REGION Network 4: Set drive objects for drive diagnostic
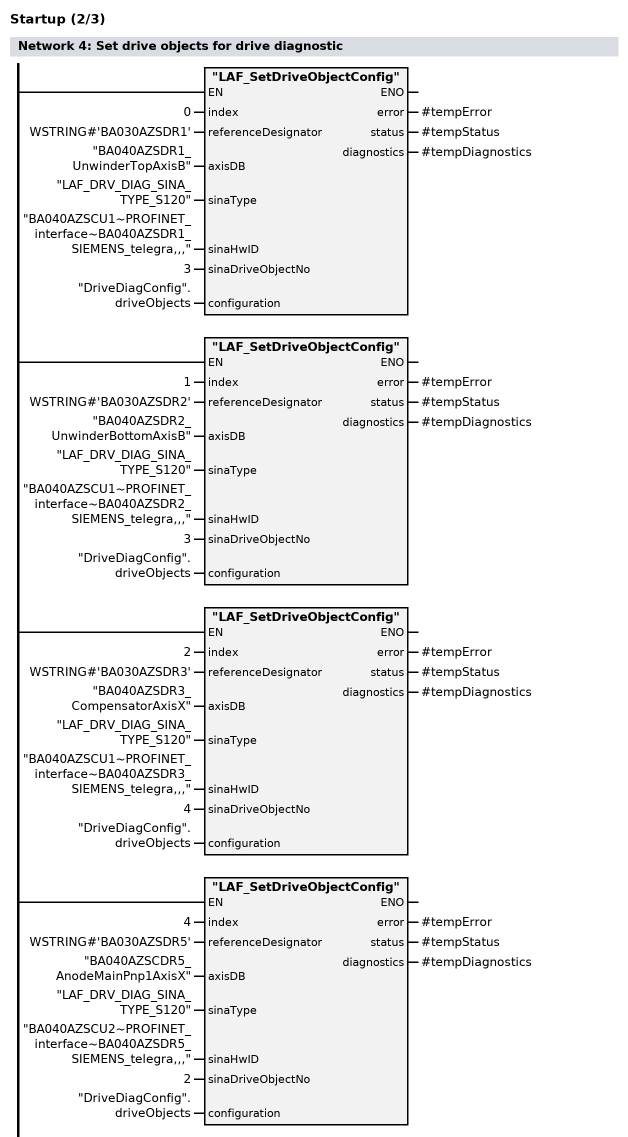
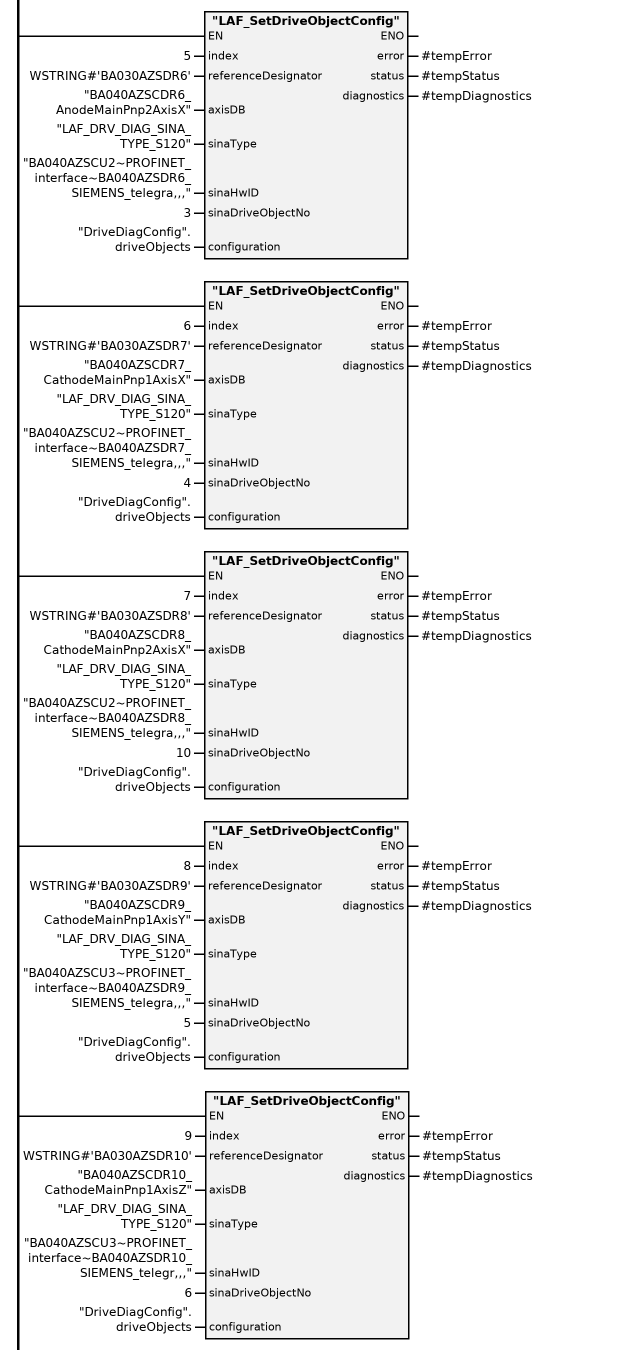
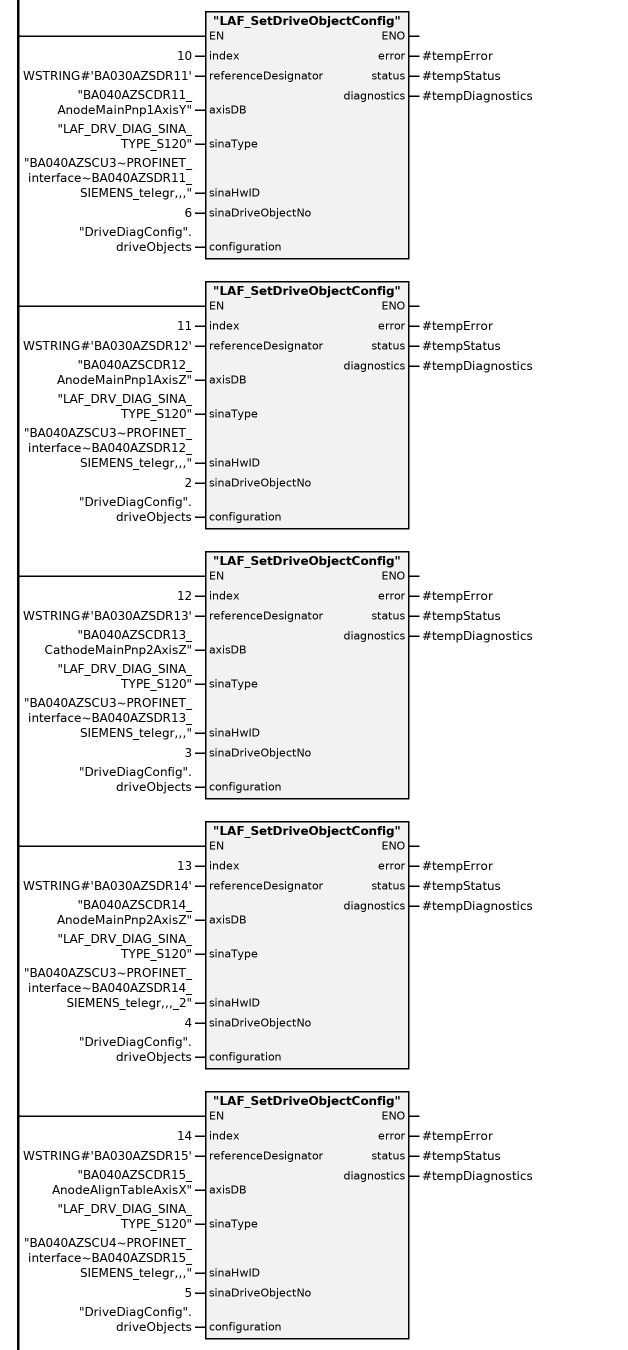
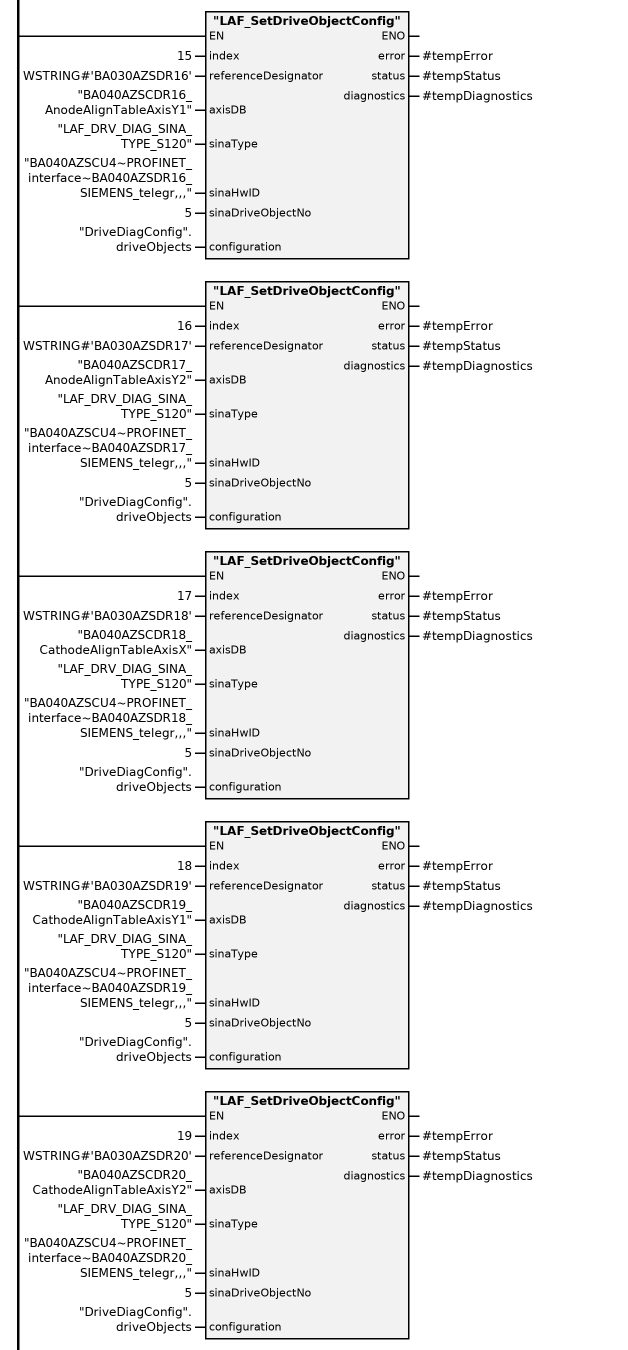
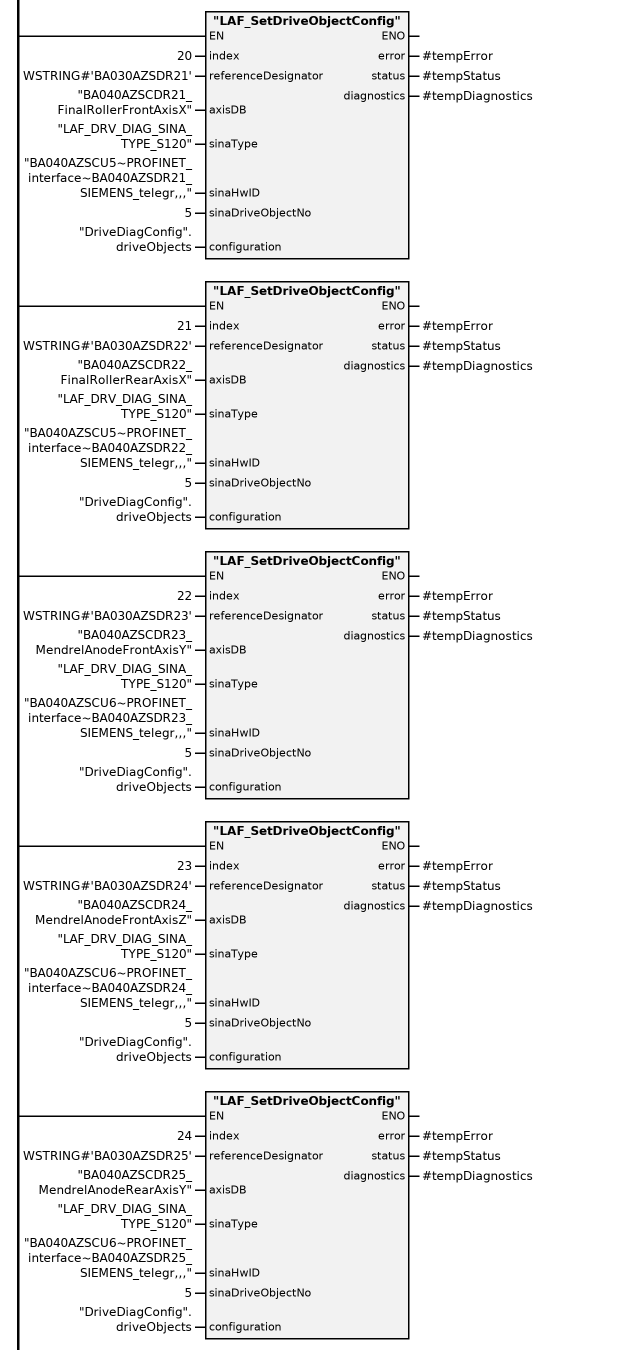
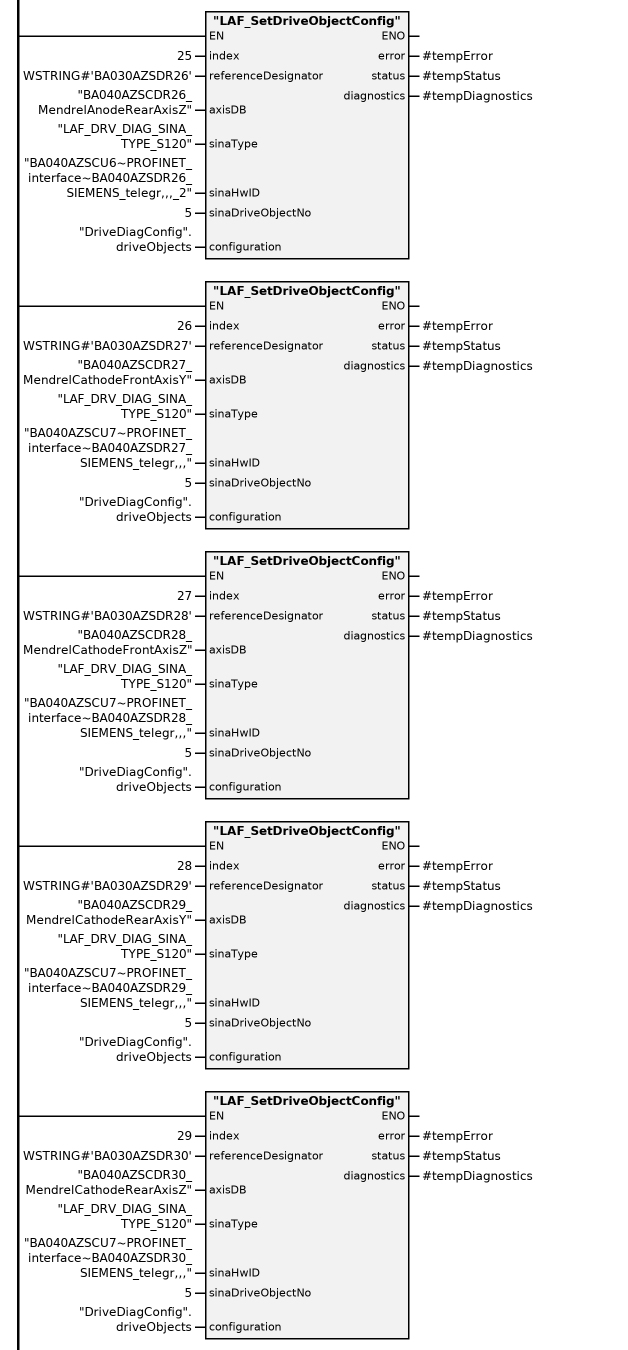
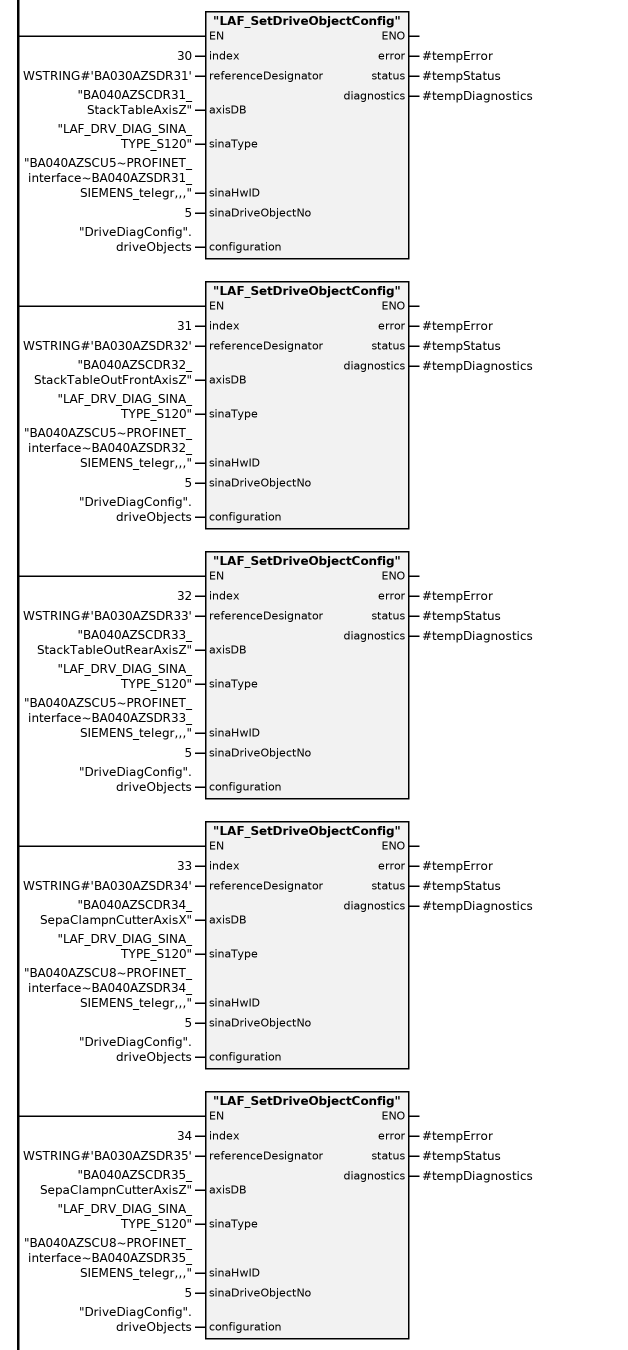
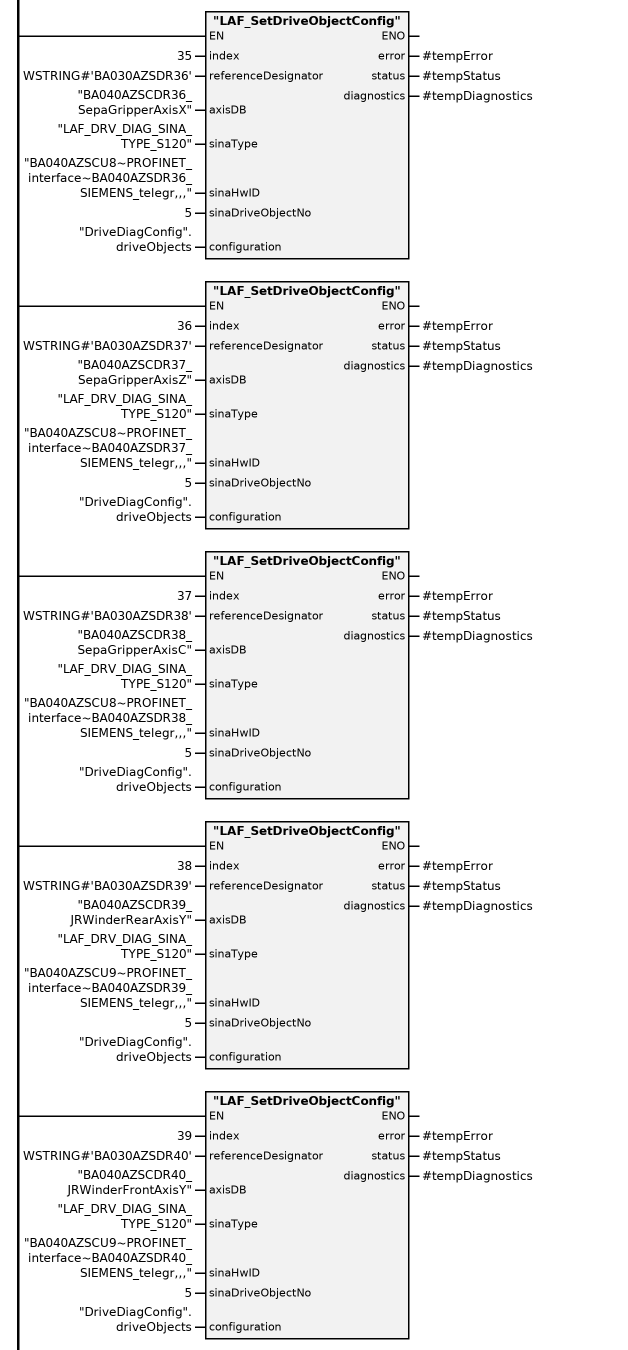
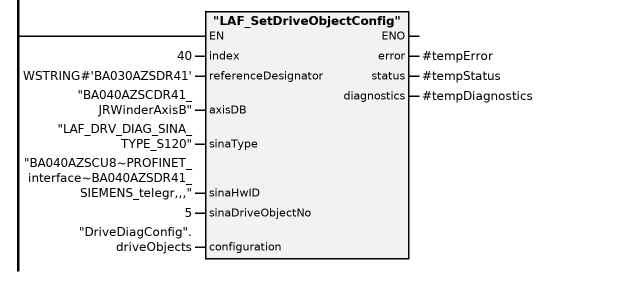
   RUNG wire#powerrail
      "LAF_SetDriveObjectConfig"(index := 0, referenceDesignator := WSTRING#'BA030AZSDR1', axisDB := "BA040AZSDR1_UnwinderTopAxisB", sinaType := "LAF_DRV_DIAG_SINA_TYPE_S120", sinaHwID := "BA040AZSCU1~PROFINET_interface~BA040AZSDR1_SIEMENS_telegra,,,", sinaDriveObjectNo := 3, configuration := "DriveDiagConfig".driveObjects, error => #tempError, status => #tempStatus, diagnostics => #tempDiagnostics)
   END_RUNG
   RUNG wire#powerrail
      "LAF_SetDriveObjectConfig"(index := 1, referenceDesignator := WSTRING#'BA030AZSDR2', axisDB := "BA040AZSDR2_UnwinderBottomAxisB", sinaType := "LAF_DRV_DIAG_SINA_TYPE_S120", sinaHwID := "BA040AZSCU1~PROFINET_interface~BA040AZSDR2_SIEMENS_telegra,,,", sinaDriveObjectNo := 3, configuration := "DriveDiagConfig".driveObjects, error => #tempError, status => #tempStatus, diagnostics => #tempDiagnostics)
   END_RUNG
   RUNG wire#powerrail
      "LAF_SetDriveObjectConfig"(index := 2, referenceDesignator := WSTRING#'BA030AZSDR3', axisDB := "BA040AZSDR3_CompensatorAxisX", sinaType := "LAF_DRV_DIAG_SINA_TYPE_S120", sinaHwID := "BA040AZSCU1~PROFINET_interface~BA040AZSDR3_SIEMENS_telegra,,,", sinaDriveObjectNo := 4, configuration := "DriveDiagConfig".driveObjects, error => #tempError, status => #tempStatus, diagnostics => #tempDiagnostics)
   END_RUNG
   RUNG wire#powerrail
      "LAF_SetDriveObjectConfig"(index := 4, referenceDesignator := WSTRING#'BA030AZSDR5', axisDB := "BA040AZSCDR5_AnodeMainPnp1AxisX", sinaType := "LAF_DRV_DIAG_SINA_TYPE_S120", sinaHwID := "BA040AZSCU2~PROFINET_interface~BA040AZSDR5_SIEMENS_telegra,,,", sinaDriveObjectNo := 2, configuration := "DriveDiagConfig".driveObjects, error => #tempError, status => #tempStatus, diagnostics => #tempDiagnostics)
   END_RUNG
   RUNG wire#powerrail
      "LAF_SetDriveObjectConfig"(index := 5, referenceDesignator := WSTRING#'BA030AZSDR6', axisDB := "BA040AZSCDR6_AnodeMainPnp2AxisX", sinaType := "LAF_DRV_DIAG_SINA_TYPE_S120", sinaHwID := "BA040AZSCU2~PROFINET_interface~BA040AZSDR6_SIEMENS_telegra,,,", sinaDriveObjectNo := 3, configuration := "DriveDiagConfig".driveObjects, error => #tempError, status => #tempStatus, diagnostics => #tempDiagnostics)
   END_RUNG
   RUNG wire#powerrail
      "LAF_SetDriveObjectConfig"(index := 6, referenceDesignator := WSTRING#'BA030AZSDR7', axisDB := "BA040AZSCDR7_CathodeMainPnp1AxisX", sinaType := "LAF_DRV_DIAG_SINA_TYPE_S120", sinaHwID := "BA040AZSCU2~PROFINET_interface~BA040AZSDR7_SIEMENS_telegra,,,", sinaDriveObjectNo := 4, configuration := "DriveDiagConfig".driveObjects, error => #tempError, status => #tempStatus, diagnostics => #tempDiagnostics)
   END_RUNG
   RUNG wire#powerrail
      "LAF_SetDriveObjectConfig"(index := 7, referenceDesignator := WSTRING#'BA030AZSDR8', axisDB := "BA040AZSCDR8_CathodeMainPnp2AxisX", sinaType := "LAF_DRV_DIAG_SINA_TYPE_S120", sinaHwID := "BA040AZSCU2~PROFINET_interface~BA040AZSDR8_SIEMENS_telegra,,,", sinaDriveObjectNo := 10, configuration := "DriveDiagConfig".driveObjects, error => #tempError, status => #tempStatus, diagnostics => #tempDiagnostics)
   END_RUNG
   RUNG wire#powerrail
      "LAF_SetDriveObjectConfig"(index := 8, referenceDesignator := WSTRING#'BA030AZSDR9', axisDB := "BA040AZSCDR9_CathodeMainPnp1AxisY", sinaType := "LAF_DRV_DIAG_SINA_TYPE_S120", sinaHwID := "BA040AZSCU3~PROFINET_interface~BA040AZSDR9_SIEMENS_telegra,,,", sinaDriveObjectNo := 5, configuration := "DriveDiagConfig".driveObjects, error => #tempError, status => #tempStatus, diagnostics => #tempDiagnostics)
   END_RUNG
   RUNG wire#powerrail
      "LAF_SetDriveObjectConfig"(index := 9, referenceDesignator := WSTRING#'BA030AZSDR10', axisDB := "BA040AZSCDR10_CathodeMainPnp1AxisZ", sinaType := "LAF_DRV_DIAG_SINA_TYPE_S120", sinaHwID := "BA040AZSCU3~PROFINET_interface~BA040AZSDR10_SIEMENS_telegr,,,", sinaDriveObjectNo := 6, configuration := "DriveDiagConfig".driveObjects, error => #tempError, status => #tempStatus, diagnostics => #tempDiagnostics)
   END_RUNG
   RUNG wire#powerrail
      "LAF_SetDriveObjectConfig"(index := 10, referenceDesignator := WSTRING#'BA030AZSDR11', axisDB := "BA040AZSCDR11_AnodeMainPnp1AxisY", sinaType := "LAF_DRV_DIAG_SINA_TYPE_S120", sinaHwID := "BA040AZSCU3~PROFINET_interface~BA040AZSDR11_SIEMENS_telegr,,,", sinaDriveObjectNo := 6, configuration := "DriveDiagConfig".driveObjects, error => #tempError, status => #tempStatus, diagnostics => #tempDiagnostics)
   END_RUNG
   RUNG wire#powerrail
      "LAF_SetDriveObjectConfig"(index := 11, referenceDesignator := WSTRING#'BA030AZSDR12', axisDB := "BA040AZSCDR12_AnodeMainPnp1AxisZ", sinaType := "LAF_DRV_DIAG_SINA_TYPE_S120", sinaHwID := "BA040AZSCU3~PROFINET_interface~BA040AZSDR12_SIEMENS_telegr,,,", sinaDriveObjectNo := 2, configuration := "DriveDiagConfig".driveObjects, error => #tempError, status => #tempStatus, diagnostics => #tempDiagnostics)
   END_RUNG
   RUNG wire#powerrail
      "LAF_SetDriveObjectConfig"(index := 12, referenceDesignator := WSTRING#'BA030AZSDR13', axisDB := "BA040AZSCDR13_CathodeMainPnp2AxisZ", sinaType := "LAF_DRV_DIAG_SINA_TYPE_S120", sinaHwID := "BA040AZSCU3~PROFINET_interface~BA040AZSDR13_SIEMENS_telegr,,,", sinaDriveObjectNo := 3, configuration := "DriveDiagConfig".driveObjects, error => #tempError, status => #tempStatus, diagnostics => #tempDiagnostics)
   END_RUNG
   RUNG wire#powerrail
      "LAF_SetDriveObjectConfig"(index := 13, referenceDesignator := WSTRING#'BA030AZSDR14', axisDB := "BA040AZSCDR14_AnodeMainPnp2AxisZ", sinaType := "LAF_DRV_DIAG_SINA_TYPE_S120", sinaHwID := "BA040AZSCU3~PROFINET_interface~BA040AZSDR14_SIEMENS_telegr,,,_2", sinaDriveObjectNo := 4, configuration := "DriveDiagConfig".driveObjects, error => #tempError, status => #tempStatus, diagnostics => #tempDiagnostics)
   END_RUNG
   RUNG wire#powerrail
      "LAF_SetDriveObjectConfig"(index := 14, referenceDesignator := WSTRING#'BA030AZSDR15', axisDB := "BA040AZSCDR15_AnodeAlignTableAxisX", sinaType := "LAF_DRV_DIAG_SINA_TYPE_S120", sinaHwID := "BA040AZSCU4~PROFINET_interface~BA040AZSDR15_SIEMENS_telegr,,,", sinaDriveObjectNo := 5, configuration := "DriveDiagConfig".driveObjects, error => #tempError, status => #tempStatus, diagnostics => #tempDiagnostics)
   END_RUNG
   RUNG wire#powerrail
      "LAF_SetDriveObjectConfig"(index := 15, referenceDesignator := WSTRING#'BA030AZSDR16', axisDB := "BA040AZSCDR16_AnodeAlignTableAxisY1", sinaType := "LAF_DRV_DIAG_SINA_TYPE_S120", sinaHwID := "BA040AZSCU4~PROFINET_interface~BA040AZSDR16_SIEMENS_telegr,,,", sinaDriveObjectNo := 5, configuration := "DriveDiagConfig".driveObjects, error => #tempError, status => #tempStatus, diagnostics => #tempDiagnostics)
   END_RUNG
   RUNG wire#powerrail
      "LAF_SetDriveObjectConfig"(index := 16, referenceDesignator := WSTRING#'BA030AZSDR17', axisDB := "BA040AZSCDR17_AnodeAlignTableAxisY2", sinaType := "LAF_DRV_DIAG_SINA_TYPE_S120", sinaHwID := "BA040AZSCU4~PROFINET_interface~BA040AZSDR17_SIEMENS_telegr,,,", sinaDriveObjectNo := 5, configuration := "DriveDiagConfig".driveObjects, error => #tempError, status => #tempStatus, diagnostics => #tempDiagnostics)
   END_RUNG
   RUNG wire#powerrail
      "LAF_SetDriveObjectConfig"(index := 17, referenceDesignator := WSTRING#'BA030AZSDR18', axisDB := "BA040AZSCDR18_CathodeAlignTableAxisX", sinaType := "LAF_DRV_DIAG_SINA_TYPE_S120", sinaHwID := "BA040AZSCU4~PROFINET_interface~BA040AZSDR18_SIEMENS_telegr,,,", sinaDriveObjectNo := 5, configuration := "DriveDiagConfig".driveObjects, error => #tempError, status => #tempStatus, diagnostics => #tempDiagnostics)
   END_RUNG
   RUNG wire#powerrail
      "LAF_SetDriveObjectConfig"(index := 18, referenceDesignator := WSTRING#'BA030AZSDR19', axisDB := "BA040AZSCDR19_CathodeAlignTableAxisY1", sinaType := "LAF_DRV_DIAG_SINA_TYPE_S120", sinaHwID := "BA040AZSCU4~PROFINET_interface~BA040AZSDR19_SIEMENS_telegr,,,", sinaDriveObjectNo := 5, configuration := "DriveDiagConfig".driveObjects, error => #tempError, status => #tempStatus, diagnostics => #tempDiagnostics)
   END_RUNG
   RUNG wire#powerrail
      "LAF_SetDriveObjectConfig"(index := 19, referenceDesignator := WSTRING#'BA030AZSDR20', axisDB := "BA040AZSCDR20_CathodeAlignTableAxisY2", sinaType := "LAF_DRV_DIAG_SINA_TYPE_S120", sinaHwID := "BA040AZSCU4~PROFINET_interface~BA040AZSDR20_SIEMENS_telegr,,,", sinaDriveObjectNo := 5, configuration := "DriveDiagConfig".driveObjects, error => #tempError, status => #tempStatus, diagnostics => #tempDiagnostics)
   END_RUNG
   RUNG wire#powerrail
      "LAF_SetDriveObjectConfig"(index := 20, referenceDesignator := WSTRING#'BA030AZSDR21', axisDB := "BA040AZSCDR21_FinalRollerFrontAxisX", sinaType := "LAF_DRV_DIAG_SINA_TYPE_S120", sinaHwID := "BA040AZSCU5~PROFINET_interface~BA040AZSDR21_SIEMENS_telegr,,,", sinaDriveObjectNo := 5, configuration := "DriveDiagConfig".driveObjects, error => #tempError, status => #tempStatus, diagnostics => #tempDiagnostics)
   END_RUNG
   RUNG wire#powerrail
      "LAF_SetDriveObjectConfig"(index := 21, referenceDesignator := WSTRING#'BA030AZSDR22', axisDB := "BA040AZSCDR22_FinalRollerRearAxisX", sinaType := "LAF_DRV_DIAG_SINA_TYPE_S120", sinaHwID := "BA040AZSCU5~PROFINET_interface~BA040AZSDR22_SIEMENS_telegr,,,", sinaDriveObjectNo := 5, configuration := "DriveDiagConfig".driveObjects, error => #tempError, status => #tempStatus, diagnostics => #tempDiagnostics)
   END_RUNG
   RUNG wire#powerrail
      "LAF_SetDriveObjectConfig"(index := 22, referenceDesignator := WSTRING#'BA030AZSDR23', axisDB := "BA040AZSCDR23_MendrelAnodeFrontAxisY", sinaType := "LAF_DRV_DIAG_SINA_TYPE_S120", sinaHwID := "BA040AZSCU6~PROFINET_interface~BA040AZSDR23_SIEMENS_telegr,,,", sinaDriveObjectNo := 5, configuration := "DriveDiagConfig".driveObjects, error => #tempError, status => #tempStatus, diagnostics => #tempDiagnostics)
   END_RUNG
   RUNG wire#powerrail
      "LAF_SetDriveObjectConfig"(index := 23, referenceDesignator := WSTRING#'BA030AZSDR24', axisDB := "BA040AZSCDR24_MendrelAnodeFrontAxisZ", sinaType := "LAF_DRV_DIAG_SINA_TYPE_S120", sinaHwID := "BA040AZSCU6~PROFINET_interface~BA040AZSDR24_SIEMENS_telegr,,,", sinaDriveObjectNo := 5, configuration := "DriveDiagConfig".driveObjects, error => #tempError, status => #tempStatus, diagnostics => #tempDiagnostics)
   END_RUNG
   RUNG wire#powerrail
      "LAF_SetDriveObjectConfig"(index := 24, referenceDesignator := WSTRING#'BA030AZSDR25', axisDB := "BA040AZSCDR25_MendrelAnodeRearAxisY", sinaType := "LAF_DRV_DIAG_SINA_TYPE_S120", sinaHwID := "BA040AZSCU6~PROFINET_interface~BA040AZSDR25_SIEMENS_telegr,,,", sinaDriveObjectNo := 5, configuration := "DriveDiagConfig".driveObjects, error => #tempError, status => #tempStatus, diagnostics => #tempDiagnostics)
   END_RUNG
   RUNG wire#powerrail
      "LAF_SetDriveObjectConfig"(index := 25, referenceDesignator := WSTRING#'BA030AZSDR26', axisDB := "BA040AZSCDR26_MendrelAnodeRearAxisZ", sinaType := "LAF_DRV_DIAG_SINA_TYPE_S120", sinaHwID := "BA040AZSCU6~PROFINET_interface~BA040AZSDR26_SIEMENS_telegr,,,_2", sinaDriveObjectNo := 5, configuration := "DriveDiagConfig".driveObjects, error => #tempError, status => #tempStatus, diagnostics => #tempDiagnostics)
   END_RUNG
   RUNG wire#powerrail
      "LAF_SetDriveObjectConfig"(index := 26, referenceDesignator := WSTRING#'BA030AZSDR27', axisDB := "BA040AZSCDR27_MendrelCathodeFrontAxisY", sinaType := "LAF_DRV_DIAG_SINA_TYPE_S120", sinaHwID := "BA040AZSCU7~PROFINET_interface~BA040AZSDR27_SIEMENS_telegr,,,", sinaDriveObjectNo := 5, configuration := "DriveDiagConfig".driveObjects, error => #tempError, status => #tempStatus, diagnostics => #tempDiagnostics)
   END_RUNG
   RUNG wire#powerrail
      "LAF_SetDriveObjectConfig"(index := 27, referenceDesignator := WSTRING#'BA030AZSDR28', axisDB := "BA040AZSCDR28_MendrelCathodeFrontAxisZ", sinaType := "LAF_DRV_DIAG_SINA_TYPE_S120", sinaHwID := "BA040AZSCU7~PROFINET_interface~BA040AZSDR28_SIEMENS_telegr,,,", sinaDriveObjectNo := 5, configuration := "DriveDiagConfig".driveObjects, error => #tempError, status => #tempStatus, diagnostics => #tempDiagnostics)
   END_RUNG
   RUNG wire#powerrail
      "LAF_SetDriveObjectConfig"(index := 28, referenceDesignator := WSTRING#'BA030AZSDR29', axisDB := "BA040AZSCDR29_MendrelCathodeRearAxisY", sinaType := "LAF_DRV_DIAG_SINA_TYPE_S120", sinaHwID := "BA040AZSCU7~PROFINET_interface~BA040AZSDR29_SIEMENS_telegr,,,", sinaDriveObjectNo := 5, configuration := "DriveDiagConfig".driveObjects, error => #tempError, status => #tempStatus, diagnostics => #tempDiagnostics)
   END_RUNG
   RUNG wire#powerrail
      "LAF_SetDriveObjectConfig"(index := 29, referenceDesignator := WSTRING#'BA030AZSDR30', axisDB := "BA040AZSCDR30_MendrelCathodeRearAxisZ", sinaType := "LAF_DRV_DIAG_SINA_TYPE_S120", sinaHwID := "BA040AZSCU7~PROFINET_interface~BA040AZSDR30_SIEMENS_telegr,,,", sinaDriveObjectNo := 5, configuration := "DriveDiagConfig".driveObjects, error => #tempError, status => #tempStatus, diagnostics => #tempDiagnostics)
   END_RUNG
   RUNG wire#powerrail
      "LAF_SetDriveObjectConfig"(index := 30, referenceDesignator := WSTRING#'BA030AZSDR31', axisDB := "BA040AZSCDR31_StackTableAxisZ", sinaType := "LAF_DRV_DIAG_SINA_TYPE_S120", sinaHwID := "BA040AZSCU5~PROFINET_interface~BA040AZSDR31_SIEMENS_telegr,,,", sinaDriveObjectNo := 5, configuration := "DriveDiagConfig".driveObjects, error => #tempError, status => #tempStatus, diagnostics => #tempDiagnostics)
   END_RUNG
   RUNG wire#powerrail
      "LAF_SetDriveObjectConfig"(index := 31, referenceDesignator := WSTRING#'BA030AZSDR32', axisDB := "BA040AZSCDR32_StackTableOutFrontAxisZ", sinaType := "LAF_DRV_DIAG_SINA_TYPE_S120", sinaHwID := "BA040AZSCU5~PROFINET_interface~BA040AZSDR32_SIEMENS_telegr,,,", sinaDriveObjectNo := 5, configuration := "DriveDiagConfig".driveObjects, error => #tempError, status => #tempStatus, diagnostics => #tempDiagnostics)
   END_RUNG
   RUNG wire#powerrail
      "LAF_SetDriveObjectConfig"(index := 32, referenceDesignator := WSTRING#'BA030AZSDR33', axisDB := "BA040AZSCDR33_StackTableOutRearAxisZ", sinaType := "LAF_DRV_DIAG_SINA_TYPE_S120", sinaHwID := "BA040AZSCU5~PROFINET_interface~BA040AZSDR33_SIEMENS_telegr,,,", sinaDriveObjectNo := 5, configuration := "DriveDiagConfig".driveObjects, error => #tempError, status => #tempStatus, diagnostics => #tempDiagnostics)
   END_RUNG
   RUNG wire#powerrail
      "LAF_SetDriveObjectConfig"(index := 33, referenceDesignator := WSTRING#'BA030AZSDR34', axisDB := "BA040AZSCDR34_SepaClampnCutterAxisX", sinaType := "LAF_DRV_DIAG_SINA_TYPE_S120", sinaHwID := "BA040AZSCU8~PROFINET_interface~BA040AZSDR34_SIEMENS_telegr,,,", sinaDriveObjectNo := 5, configuration := "DriveDiagConfig".driveObjects, error => #tempError, status => #tempStatus, diagnostics => #tempDiagnostics)
   END_RUNG
   RUNG wire#powerrail
      "LAF_SetDriveObjectConfig"(index := 34, referenceDesignator := WSTRING#'BA030AZSDR35', axisDB := "BA040AZSCDR35_SepaClampnCutterAxisZ", sinaType := "LAF_DRV_DIAG_SINA_TYPE_S120", sinaHwID := "BA040AZSCU8~PROFINET_interface~BA040AZSDR35_SIEMENS_telegr,,,", sinaDriveObjectNo := 5, configuration := "DriveDiagConfig".driveObjects, error => #tempError, status => #tempStatus, diagnostics => #tempDiagnostics)
   END_RUNG
   RUNG wire#powerrail
      "LAF_SetDriveObjectConfig"(index := 35, referenceDesignator := WSTRING#'BA030AZSDR36', axisDB := "BA040AZSCDR36_SepaGripperAxisX", sinaType := "LAF_DRV_DIAG_SINA_TYPE_S120", sinaHwID := "BA040AZSCU8~PROFINET_interface~BA040AZSDR36_SIEMENS_telegr,,,", sinaDriveObjectNo := 5, configuration := "DriveDiagConfig".driveObjects, error => #tempError, status => #tempStatus, diagnostics => #tempDiagnostics)
   END_RUNG
   RUNG wire#powerrail
      "LAF_SetDriveObjectConfig"(index := 36, referenceDesignator := WSTRING#'BA030AZSDR37', axisDB := "BA040AZSCDR37_SepaGripperAxisZ", sinaType := "LAF_DRV_DIAG_SINA_TYPE_S120", sinaHwID := "BA040AZSCU8~PROFINET_interface~BA040AZSDR37_SIEMENS_telegr,,,", sinaDriveObjectNo := 5, configuration := "DriveDiagConfig".driveObjects, error => #tempError, status => #tempStatus, diagnostics => #tempDiagnostics)
   END_RUNG
   RUNG wire#powerrail
      "LAF_SetDriveObjectConfig"(index := 37, referenceDesignator := WSTRING#'BA030AZSDR38', axisDB := "BA040AZSCDR38_SepaGripperAxisC", sinaType := "LAF_DRV_DIAG_SINA_TYPE_S120", sinaHwID := "BA040AZSCU8~PROFINET_interface~BA040AZSDR38_SIEMENS_telegr,,,", sinaDriveObjectNo := 5, configuration := "DriveDiagConfig".driveObjects, error => #tempError, status => #tempStatus, diagnostics => #tempDiagnostics)
   END_RUNG
   RUNG wire#powerrail
      "LAF_SetDriveObjectConfig"(index := 38, referenceDesignator := WSTRING#'BA030AZSDR39', axisDB := "BA040AZSCDR39_JRWinderRearAxisY", sinaType := "LAF_DRV_DIAG_SINA_TYPE_S120", sinaHwID := "BA040AZSCU9~PROFINET_interface~BA040AZSDR39_SIEMENS_telegr,,,", sinaDriveObjectNo := 5, configuration := "DriveDiagConfig".driveObjects, error => #tempError, status => #tempStatus, diagnostics => #tempDiagnostics)
   END_RUNG
   RUNG wire#powerrail
      "LAF_SetDriveObjectConfig"(index := 39, referenceDesignator := WSTRING#'BA030AZSDR40', axisDB := "BA040AZSCDR40_JRWinderFrontAxisY", sinaType := "LAF_DRV_DIAG_SINA_TYPE_S120", sinaHwID := "BA040AZSCU9~PROFINET_interface~BA040AZSDR40_SIEMENS_telegr,,,", sinaDriveObjectNo := 5, configuration := "DriveDiagConfig".driveObjects, error => #tempError, status => #tempStatus, diagnostics => #tempDiagnostics)
   END_RUNG
   RUNG wire#powerrail
      "LAF_SetDriveObjectConfig"(index := 40, referenceDesignator := WSTRING#'BA030AZSDR41', axisDB := "BA040AZSCDR41_JRWinderAxisB", sinaType := "LAF_DRV_DIAG_SINA_TYPE_S120", sinaHwID := "BA040AZSCU8~PROFINET_interface~BA040AZSDR41_SIEMENS_telegr,,,", sinaDriveObjectNo := 5, configuration := "DriveDiagConfig".driveObjects, error => #tempError, status => #tempStatus, diagnostics => #tempDiagnostics)
   END_RUNG
   // the same network as SCL:
   "LAF_SetDriveObjectConfig"(index := 0,
                           referenceDesignator := WSTRING#'BA030AZSDR1',
                           axisDB := "BA040AZSDR1_UnwinderTopAxisB",
                           sinaType := "LAF_DRV_DIAG_SINA_TYPE_S120",
                           sinaHwID := "BA040AZSCU1~PROFINET_interface~BA040AZSDR1_SIEMENS_telegra,,,",
                           sinaDriveObjectNo := 3,
                           configuration := "DriveDiagConfig".driveObjects,
                           error => #tempError,
                           status => #tempStatus,
                           diagnostics => #tempDiagnostics);
   "LAF_SetDriveObjectConfig"(index := 1,
                           referenceDesignator := WSTRING#'BA030AZSDR2',
                           axisDB := "BA040AZSDR2_UnwinderBottomAxisB",
                           sinaType := "LAF_DRV_DIAG_SINA_TYPE_S120",
                           sinaHwID := "BA040AZSCU1~PROFINET_interface~BA040AZSDR2_SIEMENS_telegra,,,",
                           sinaDriveObjectNo := 3,
                           configuration := "DriveDiagConfig".driveObjects,
                           error => #tempError,
                           status => #tempStatus,
                           diagnostics => #tempDiagnostics);
   "LAF_SetDriveObjectConfig"(index := 2,
                           referenceDesignator := WSTRING#'BA030AZSDR3',
                           axisDB := "BA040AZSDR3_CompensatorAxisX",
                           sinaType := "LAF_DRV_DIAG_SINA_TYPE_S120",
                           sinaHwID := "BA040AZSCU1~PROFINET_interface~BA040AZSDR3_SIEMENS_telegra,,,",
                           sinaDriveObjectNo := 4,
                           configuration := "DriveDiagConfig".driveObjects,
                           error => #tempError,
                           status => #tempStatus,
                           diagnostics => #tempDiagnostics);
   "LAF_SetDriveObjectConfig"(index := 4,
                           referenceDesignator := WSTRING#'BA030AZSDR5',
                           axisDB := "BA040AZSCDR5_AnodeMainPnp1AxisX",
                           sinaType := "LAF_DRV_DIAG_SINA_TYPE_S120",
                           sinaHwID := "BA040AZSCU2~PROFINET_interface~BA040AZSDR5_SIEMENS_telegra,,,",
                           sinaDriveObjectNo := 2,
                           configuration := "DriveDiagConfig".driveObjects,
                           error => #tempError,
                           status => #tempStatus,
                           diagnostics => #tempDiagnostics);
   "LAF_SetDriveObjectConfig"(index := 5,
                           referenceDesignator := WSTRING#'BA030AZSDR6',
                           axisDB := "BA040AZSCDR6_AnodeMainPnp2AxisX",
                           sinaType := "LAF_DRV_DIAG_SINA_TYPE_S120",
                           sinaHwID := "BA040AZSCU2~PROFINET_interface~BA040AZSDR6_SIEMENS_telegra,,,",
                           sinaDriveObjectNo := 3,
                           configuration := "DriveDiagConfig".driveObjects,
                           error => #tempError,
                           status => #tempStatus,
                           diagnostics => #tempDiagnostics);
   "LAF_SetDriveObjectConfig"(index := 6,
                           referenceDesignator := WSTRING#'BA030AZSDR7',
                           axisDB := "BA040AZSCDR7_CathodeMainPnp1AxisX",
                           sinaType := "LAF_DRV_DIAG_SINA_TYPE_S120",
                           sinaHwID := "BA040AZSCU2~PROFINET_interface~BA040AZSDR7_SIEMENS_telegra,,,",
                           sinaDriveObjectNo := 4,
                           configuration := "DriveDiagConfig".driveObjects,
                           error => #tempError,
                           status => #tempStatus,
                           diagnostics => #tempDiagnostics);
   "LAF_SetDriveObjectConfig"(index := 7,
                           referenceDesignator := WSTRING#'BA030AZSDR8',
                           axisDB := "BA040AZSCDR8_CathodeMainPnp2AxisX",
                           sinaType := "LAF_DRV_DIAG_SINA_TYPE_S120",
                           sinaHwID := "BA040AZSCU2~PROFINET_interface~BA040AZSDR8_SIEMENS_telegra,,,",
                           sinaDriveObjectNo := 10,
                           configuration := "DriveDiagConfig".driveObjects,
                           error => #tempError,
                           status => #tempStatus,
                           diagnostics => #tempDiagnostics);
   "LAF_SetDriveObjectConfig"(index := 8,
                           referenceDesignator := WSTRING#'BA030AZSDR9',
                           axisDB := "BA040AZSCDR9_CathodeMainPnp1AxisY",
                           sinaType := "LAF_DRV_DIAG_SINA_TYPE_S120",
                           sinaHwID := "BA040AZSCU3~PROFINET_interface~BA040AZSDR9_SIEMENS_telegra,,,",
                           sinaDriveObjectNo := 5,
                           configuration := "DriveDiagConfig".driveObjects,
                           error => #tempError,
                           status => #tempStatus,
                           diagnostics => #tempDiagnostics);
   "LAF_SetDriveObjectConfig"(index := 9,
                           referenceDesignator := WSTRING#'BA030AZSDR10',
                           axisDB := "BA040AZSCDR10_CathodeMainPnp1AxisZ",
                           sinaType := "LAF_DRV_DIAG_SINA_TYPE_S120",
                           sinaHwID := "BA040AZSCU3~PROFINET_interface~BA040AZSDR10_SIEMENS_telegr,,,",
                           sinaDriveObjectNo := 6,
                           configuration := "DriveDiagConfig".driveObjects,
                           error => #tempError,
                           status => #tempStatus,
                           diagnostics => #tempDiagnostics);
   "LAF_SetDriveObjectConfig"(index := 10,
                           referenceDesignator := WSTRING#'BA030AZSDR11',
                           axisDB := "BA040AZSCDR11_AnodeMainPnp1AxisY",
                           sinaType := "LAF_DRV_DIAG_SINA_TYPE_S120",
                           sinaHwID := "BA040AZSCU3~PROFINET_interface~BA040AZSDR11_SIEMENS_telegr,,,",
                           sinaDriveObjectNo := 6,
                           configuration := "DriveDiagConfig".driveObjects,
                           error => #tempError,
                           status => #tempStatus,
                           diagnostics => #tempDiagnostics);
   "LAF_SetDriveObjectConfig"(index := 11,
                           referenceDesignator := WSTRING#'BA030AZSDR12',
                           axisDB := "BA040AZSCDR12_AnodeMainPnp1AxisZ",
                           sinaType := "LAF_DRV_DIAG_SINA_TYPE_S120",
                           sinaHwID := "BA040AZSCU3~PROFINET_interface~BA040AZSDR12_SIEMENS_telegr,,,",
                           sinaDriveObjectNo := 2,
                           configuration := "DriveDiagConfig".driveObjects,
                           error => #tempError,
                           status => #tempStatus,
                           diagnostics => #tempDiagnostics);
   "LAF_SetDriveObjectConfig"(index := 12,
                           referenceDesignator := WSTRING#'BA030AZSDR13',
                           axisDB := "BA040AZSCDR13_CathodeMainPnp2AxisZ",
                           sinaType := "LAF_DRV_DIAG_SINA_TYPE_S120",
                           sinaHwID := "BA040AZSCU3~PROFINET_interface~BA040AZSDR13_SIEMENS_telegr,,,",
                           sinaDriveObjectNo := 3,
                           configuration := "DriveDiagConfig".driveObjects,
                           error => #tempError,
                           status => #tempStatus,
                           diagnostics => #tempDiagnostics);
   "LAF_SetDriveObjectConfig"(index := 13,
                           referenceDesignator := WSTRING#'BA030AZSDR14',
                           axisDB := "BA040AZSCDR14_AnodeMainPnp2AxisZ",
                           sinaType := "LAF_DRV_DIAG_SINA_TYPE_S120",
                           sinaHwID := "BA040AZSCU3~PROFINET_interface~BA040AZSDR14_SIEMENS_telegr,,,_2",
                           sinaDriveObjectNo := 4,
                           configuration := "DriveDiagConfig".driveObjects,
                           error => #tempError,
                           status => #tempStatus,
                           diagnostics => #tempDiagnostics);
   "LAF_SetDriveObjectConfig"(index := 14,
                           referenceDesignator := WSTRING#'BA030AZSDR15',
                           axisDB := "BA040AZSCDR15_AnodeAlignTableAxisX",
                           sinaType := "LAF_DRV_DIAG_SINA_TYPE_S120",
                           sinaHwID := "BA040AZSCU4~PROFINET_interface~BA040AZSDR15_SIEMENS_telegr,,,",
                           sinaDriveObjectNo := 5,
                           configuration := "DriveDiagConfig".driveObjects,
                           error => #tempError,
                           status => #tempStatus,
                           diagnostics => #tempDiagnostics);
   "LAF_SetDriveObjectConfig"(index := 15,
                           referenceDesignator := WSTRING#'BA030AZSDR16',
                           axisDB := "BA040AZSCDR16_AnodeAlignTableAxisY1",
                           sinaType := "LAF_DRV_DIAG_SINA_TYPE_S120",
                           sinaHwID := "BA040AZSCU4~PROFINET_interface~BA040AZSDR16_SIEMENS_telegr,,,",
                           sinaDriveObjectNo := 5,
                           configuration := "DriveDiagConfig".driveObjects,
                           error => #tempError,
                           status => #tempStatus,
                           diagnostics => #tempDiagnostics);
   "LAF_SetDriveObjectConfig"(index := 16,
                           referenceDesignator := WSTRING#'BA030AZSDR17',
                           axisDB := "BA040AZSCDR17_AnodeAlignTableAxisY2",
                           sinaType := "LAF_DRV_DIAG_SINA_TYPE_S120",
                           sinaHwID := "BA040AZSCU4~PROFINET_interface~BA040AZSDR17_SIEMENS_telegr,,,",
                           sinaDriveObjectNo := 5,
                           configuration := "DriveDiagConfig".driveObjects,
                           error => #tempError,
                           status => #tempStatus,
                           diagnostics => #tempDiagnostics);
   "LAF_SetDriveObjectConfig"(index := 17,
                           referenceDesignator := WSTRING#'BA030AZSDR18',
                           axisDB := "BA040AZSCDR18_CathodeAlignTableAxisX",
                           sinaType := "LAF_DRV_DIAG_SINA_TYPE_S120",
                           sinaHwID := "BA040AZSCU4~PROFINET_interface~BA040AZSDR18_SIEMENS_telegr,,,",
                           sinaDriveObjectNo := 5,
                           configuration := "DriveDiagConfig".driveObjects,
                           error => #tempError,
                           status => #tempStatus,
                           diagnostics => #tempDiagnostics);
   "LAF_SetDriveObjectConfig"(index := 18,
                           referenceDesignator := WSTRING#'BA030AZSDR19',
                           axisDB := "BA040AZSCDR19_CathodeAlignTableAxisY1",
                           sinaType := "LAF_DRV_DIAG_SINA_TYPE_S120",
                           sinaHwID := "BA040AZSCU4~PROFINET_interface~BA040AZSDR19_SIEMENS_telegr,,,",
                           sinaDriveObjectNo := 5,
                           configuration := "DriveDiagConfig".driveObjects,
                           error => #tempError,
                           status => #tempStatus,
                           diagnostics => #tempDiagnostics);
   "LAF_SetDriveObjectConfig"(index := 19,
                           referenceDesignator := WSTRING#'BA030AZSDR20',
                           axisDB := "BA040AZSCDR20_CathodeAlignTableAxisY2",
                           sinaType := "LAF_DRV_DIAG_SINA_TYPE_S120",
                           sinaHwID := "BA040AZSCU4~PROFINET_interface~BA040AZSDR20_SIEMENS_telegr,,,",
                           sinaDriveObjectNo := 5,
                           configuration := "DriveDiagConfig".driveObjects,
                           error => #tempError,
                           status => #tempStatus,
                           diagnostics => #tempDiagnostics);
   "LAF_SetDriveObjectConfig"(index := 20,
                           referenceDesignator := WSTRING#'BA030AZSDR21',
                           axisDB := "BA040AZSCDR21_FinalRollerFrontAxisX",
                           sinaType := "LAF_DRV_DIAG_SINA_TYPE_S120",
                           sinaHwID := "BA040AZSCU5~PROFINET_interface~BA040AZSDR21_SIEMENS_telegr,,,",
                           sinaDriveObjectNo := 5,
                           configuration := "DriveDiagConfig".driveObjects,
                           error => #tempError,
                           status => #tempStatus,
                           diagnostics => #tempDiagnostics);
   "LAF_SetDriveObjectConfig"(index := 21,
                           referenceDesignator := WSTRING#'BA030AZSDR22',
                           axisDB := "BA040AZSCDR22_FinalRollerRearAxisX",
                           sinaType := "LAF_DRV_DIAG_SINA_TYPE_S120",
                           sinaHwID := "BA040AZSCU5~PROFINET_interface~BA040AZSDR22_SIEMENS_telegr,,,",
                           sinaDriveObjectNo := 5,
                           configuration := "DriveDiagConfig".driveObjects,
                           error => #tempError,
                           status => #tempStatus,
                           diagnostics => #tempDiagnostics);
   "LAF_SetDriveObjectConfig"(index := 22,
                           referenceDesignator := WSTRING#'BA030AZSDR23',
                           axisDB := "BA040AZSCDR23_MendrelAnodeFrontAxisY",
                           sinaType := "LAF_DRV_DIAG_SINA_TYPE_S120",
                           sinaHwID := "BA040AZSCU6~PROFINET_interface~BA040AZSDR23_SIEMENS_telegr,,,",
                           sinaDriveObjectNo := 5,
                           configuration := "DriveDiagConfig".driveObjects,
                           error => #tempError,
                           status => #tempStatus,
                           diagnostics => #tempDiagnostics);
   "LAF_SetDriveObjectConfig"(index := 23,
                           referenceDesignator := WSTRING#'BA030AZSDR24',
                           axisDB := "BA040AZSCDR24_MendrelAnodeFrontAxisZ",
                           sinaType := "LAF_DRV_DIAG_SINA_TYPE_S120",
                           sinaHwID := "BA040AZSCU6~PROFINET_interface~BA040AZSDR24_SIEMENS_telegr,,,",
                           sinaDriveObjectNo := 5,
                           configuration := "DriveDiagConfig".driveObjects,
                           error => #tempError,
                           status => #tempStatus,
                           diagnostics => #tempDiagnostics);
   "LAF_SetDriveObjectConfig"(index := 24,
                           referenceDesignator := WSTRING#'BA030AZSDR25',
                           axisDB := "BA040AZSCDR25_MendrelAnodeRearAxisY",
                           sinaType := "LAF_DRV_DIAG_SINA_TYPE_S120",
                           sinaHwID := "BA040AZSCU6~PROFINET_interface~BA040AZSDR25_SIEMENS_telegr,,,",
                           sinaDriveObjectNo := 5,
                           configuration := "DriveDiagConfig".driveObjects,
                           error => #tempError,
                           status => #tempStatus,
                           diagnostics => #tempDiagnostics);
   "LAF_SetDriveObjectConfig"(index := 25,
                           referenceDesignator := WSTRING#'BA030AZSDR26',
                           axisDB := "BA040AZSCDR26_MendrelAnodeRearAxisZ",
                           sinaType := "LAF_DRV_DIAG_SINA_TYPE_S120",
                           sinaHwID := "BA040AZSCU6~PROFINET_interface~BA040AZSDR26_SIEMENS_telegr,,,_2",
                           sinaDriveObjectNo := 5,
                           configuration := "DriveDiagConfig".driveObjects,
                           error => #tempError,
                           status => #tempStatus,
                           diagnostics => #tempDiagnostics);
   "LAF_SetDriveObjectConfig"(index := 26,
                           referenceDesignator := WSTRING#'BA030AZSDR27',
                           axisDB := "BA040AZSCDR27_MendrelCathodeFrontAxisY",
                           sinaType := "LAF_DRV_DIAG_SINA_TYPE_S120",
                           sinaHwID := "BA040AZSCU7~PROFINET_interface~BA040AZSDR27_SIEMENS_telegr,,,",
                           sinaDriveObjectNo := 5,
                           configuration := "DriveDiagConfig".driveObjects,
                           error => #tempError,
                           status => #tempStatus,
                           diagnostics => #tempDiagnostics);
   "LAF_SetDriveObjectConfig"(index := 27,
                           referenceDesignator := WSTRING#'BA030AZSDR28',
                           axisDB := "BA040AZSCDR28_MendrelCathodeFrontAxisZ",
                           sinaType := "LAF_DRV_DIAG_SINA_TYPE_S120",
                           sinaHwID := "BA040AZSCU7~PROFINET_interface~BA040AZSDR28_SIEMENS_telegr,,,",
                           sinaDriveObjectNo := 5,
                           configuration := "DriveDiagConfig".driveObjects,
                           error => #tempError,
                           status => #tempStatus,
                           diagnostics => #tempDiagnostics);
   "LAF_SetDriveObjectConfig"(index := 28,
                           referenceDesignator := WSTRING#'BA030AZSDR29',
                           axisDB := "BA040AZSCDR29_MendrelCathodeRearAxisY",
                           sinaType := "LAF_DRV_DIAG_SINA_TYPE_S120",
                           sinaHwID := "BA040AZSCU7~PROFINET_interface~BA040AZSDR29_SIEMENS_telegr,,,",
                           sinaDriveObjectNo := 5,
                           configuration := "DriveDiagConfig".driveObjects,
                           error => #tempError,
                           status => #tempStatus,
                           diagnostics => #tempDiagnostics);
   "LAF_SetDriveObjectConfig"(index := 29,
                           referenceDesignator := WSTRING#'BA030AZSDR30',
                           axisDB := "BA040AZSCDR30_MendrelCathodeRearAxisZ",
                           sinaType := "LAF_DRV_DIAG_SINA_TYPE_S120",
                           sinaHwID := "BA040AZSCU7~PROFINET_interface~BA040AZSDR30_SIEMENS_telegr,,,",
                           sinaDriveObjectNo := 5,
                           configuration := "DriveDiagConfig".driveObjects,
                           error => #tempError,
                           status => #tempStatus,
                           diagnostics => #tempDiagnostics);
   "LAF_SetDriveObjectConfig"(index := 30,
                           referenceDesignator := WSTRING#'BA030AZSDR31',
                           axisDB := "BA040AZSCDR31_StackTableAxisZ",
                           sinaType := "LAF_DRV_DIAG_SINA_TYPE_S120",
                           sinaHwID := "BA040AZSCU5~PROFINET_interface~BA040AZSDR31_SIEMENS_telegr,,,",
                           sinaDriveObjectNo := 5,
                           configuration := "DriveDiagConfig".driveObjects,
                           error => #tempError,
                           status => #tempStatus,
                           diagnostics => #tempDiagnostics);
   "LAF_SetDriveObjectConfig"(index := 31,
                           referenceDesignator := WSTRING#'BA030AZSDR32',
                           axisDB := "BA040AZSCDR32_StackTableOutFrontAxisZ",
                           sinaType := "LAF_DRV_DIAG_SINA_TYPE_S120",
                           sinaHwID := "BA040AZSCU5~PROFINET_interface~BA040AZSDR32_SIEMENS_telegr,,,",
                           sinaDriveObjectNo := 5,
                           configuration := "DriveDiagConfig".driveObjects,
                           error => #tempError,
                           status => #tempStatus,
                           diagnostics => #tempDiagnostics);
   "LAF_SetDriveObjectConfig"(index := 32,
                           referenceDesignator := WSTRING#'BA030AZSDR33',
                           axisDB := "BA040AZSCDR33_StackTableOutRearAxisZ",
                           sinaType := "LAF_DRV_DIAG_SINA_TYPE_S120",
                           sinaHwID := "BA040AZSCU5~PROFINET_interface~BA040AZSDR33_SIEMENS_telegr,,,",
                           sinaDriveObjectNo := 5,
                           configuration := "DriveDiagConfig".driveObjects,
                           error => #tempError,
                           status => #tempStatus,
                           diagnostics => #tempDiagnostics);
   "LAF_SetDriveObjectConfig"(index := 33,
                           referenceDesignator := WSTRING#'BA030AZSDR34',
                           axisDB := "BA040AZSCDR34_SepaClampnCutterAxisX",
                           sinaType := "LAF_DRV_DIAG_SINA_TYPE_S120",
                           sinaHwID := "BA040AZSCU8~PROFINET_interface~BA040AZSDR34_SIEMENS_telegr,,,",
                           sinaDriveObjectNo := 5,
                           configuration := "DriveDiagConfig".driveObjects,
                           error => #tempError,
                           status => #tempStatus,
                           diagnostics => #tempDiagnostics);
   "LAF_SetDriveObjectConfig"(index := 34,
                           referenceDesignator := WSTRING#'BA030AZSDR35',
                           axisDB := "BA040AZSCDR35_SepaClampnCutterAxisZ",
                           sinaType := "LAF_DRV_DIAG_SINA_TYPE_S120",
                           sinaHwID := "BA040AZSCU8~PROFINET_interface~BA040AZSDR35_SIEMENS_telegr,,,",
                           sinaDriveObjectNo := 5,
                           configuration := "DriveDiagConfig".driveObjects,
                           error => #tempError,
                           status => #tempStatus,
                           diagnostics => #tempDiagnostics);
   "LAF_SetDriveObjectConfig"(index := 35,
                           referenceDesignator := WSTRING#'BA030AZSDR36',
                           axisDB := "BA040AZSCDR36_SepaGripperAxisX",
                           sinaType := "LAF_DRV_DIAG_SINA_TYPE_S120",
                           sinaHwID := "BA040AZSCU8~PROFINET_interface~BA040AZSDR36_SIEMENS_telegr,,,",
                           sinaDriveObjectNo := 5,
                           configuration := "DriveDiagConfig".driveObjects,
                           error => #tempError,
                           status => #tempStatus,
                           diagnostics => #tempDiagnostics);
   "LAF_SetDriveObjectConfig"(index := 36,
                           referenceDesignator := WSTRING#'BA030AZSDR37',
                           axisDB := "BA040AZSCDR37_SepaGripperAxisZ",
                           sinaType := "LAF_DRV_DIAG_SINA_TYPE_S120",
                           sinaHwID := "BA040AZSCU8~PROFINET_interface~BA040AZSDR37_SIEMENS_telegr,,,",
                           sinaDriveObjectNo := 5,
                           configuration := "DriveDiagConfig".driveObjects,
                           error => #tempError,
                           status => #tempStatus,
                           diagnostics => #tempDiagnostics);
   "LAF_SetDriveObjectConfig"(index := 37,
                           referenceDesignator := WSTRING#'BA030AZSDR38',
                           axisDB := "BA040AZSCDR38_SepaGripperAxisC",
                           sinaType := "LAF_DRV_DIAG_SINA_TYPE_S120",
                           sinaHwID := "BA040AZSCU8~PROFINET_interface~BA040AZSDR38_SIEMENS_telegr,,,",
                           sinaDriveObjectNo := 5,
                           configuration := "DriveDiagConfig".driveObjects,
                           error => #tempError,
                           status => #tempStatus,
                           diagnostics => #tempDiagnostics);
   "LAF_SetDriveObjectConfig"(index := 38,
                           referenceDesignator := WSTRING#'BA030AZSDR39',
                           axisDB := "BA040AZSCDR39_JRWinderRearAxisY",
                           sinaType := "LAF_DRV_DIAG_SINA_TYPE_S120",
                           sinaHwID := "BA040AZSCU9~PROFINET_interface~BA040AZSDR39_SIEMENS_telegr,,,",
                           sinaDriveObjectNo := 5,
                           configuration := "DriveDiagConfig".driveObjects,
                           error => #tempError,
                           status => #tempStatus,
                           diagnostics => #tempDiagnostics);
   "LAF_SetDriveObjectConfig"(index := 39,
                           referenceDesignator := WSTRING#'BA030AZSDR40',
                           axisDB := "BA040AZSCDR40_JRWinderFrontAxisY",
                           sinaType := "LAF_DRV_DIAG_SINA_TYPE_S120",
                           sinaHwID := "BA040AZSCU9~PROFINET_interface~BA040AZSDR40_SIEMENS_telegr,,,",
                           sinaDriveObjectNo := 5,
                           configuration := "DriveDiagConfig".driveObjects,
                           error => #tempError,
                           status => #tempStatus,
                           diagnostics => #tempDiagnostics);
   "LAF_SetDriveObjectConfig"(index := 40,
                           referenceDesignator := WSTRING#'BA030AZSDR41',
                           axisDB := "BA040AZSCDR41_JRWinderAxisB",
                           sinaType := "LAF_DRV_DIAG_SINA_TYPE_S120",
                           sinaHwID := "BA040AZSCU8~PROFINET_interface~BA040AZSDR41_SIEMENS_telegr,,,",
                           sinaDriveObjectNo := 5,
                           configuration := "DriveDiagConfig".driveObjects,
                           error => #tempError,
                           status => #tempStatus,
                           diagnostics => #tempDiagnostics);
END_REGION

REGION Network 5: Manual Operation Line
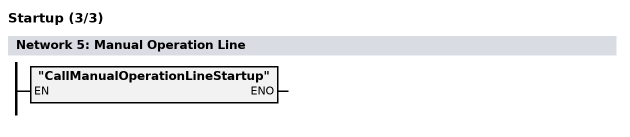
   RUNG wire#powerrail
      "CallManualOperationLineStartup"()
   END_RUNG
   // the same network as SCL:
   "CallManualOperationLineStartup"();
END_REGION
END_ORGANIZATION_BLOCK

FUNCTION "CallManualOperationLineStartup" : Void
{ S7_Optimized_Access := 'TRUE' ; Published := 'FALSE' }
VERSION : 0.1

BEGIN
	REGION Description
	(*
	    Startup call to set the configuration of the Manual Operation Line for the Equipment modules
	*)
	    
	END_REGION
	
	"LAF_InternalManual".emsWithManualOpConfigured.maxNoOfEms := "NO_OF_EM";
	
	REGION Unit 1 Equipment Module 0 configuration
	    "ManualOperationControl_U1Em0".manualOperationEm.equipmentModuleNum := 1010;
	    "ManualOperationControl_U1Em0".manualOperationEmArea[2].displayedLines := '6;';
	    "ManualOperationControl_U1Em0".manualOperationEmArea[1].displayedLines := '21;';
	END_REGION
	
	REGION Unit 1 Equipment Module 1 configuration
	    "ManualOperationControl_U1Em1".manualOperationEm.equipmentModuleNum := 1020;
	    "ManualOperationControl_U1Em1".manualOperationEmArea[2].displayedLines := '6;';
	    "ManualOperationControl_U1Em1".manualOperationEmArea[1].displayedLines := '21;';
	END_REGION
	
	REGION Unit 1 Equipment Module 2 configuration
	    "ManualOperationControl_U1Em2".manualOperationEm.equipmentModuleNum := 1030;
	    "ManualOperationControl_U1Em2".manualOperationEmArea[2].displayedLines := '1;';
	    "ManualOperationControl_U1Em2".manualOperationEmArea[1].displayedLines := '21-33;';
	END_REGION
	
	REGION Unit 1 Equipment Module 3 configuration
	    "ManualOperationControl_U1Em3".manualOperationEm.equipmentModuleNum := 1040;
	    "ManualOperationControl_U1Em3".manualOperationEmArea[2].displayedLines := '6-7;';
	    "ManualOperationControl_U1Em3".manualOperationEmArea[1].displayedLines := '21-24;';
	END_REGION
	
	REGION Unit 1 Equipment Module 4 configuration
	    "ManualOperationControl_U1Em4".manualOperationEm.equipmentModuleNum := 1050;
	    "ManualOperationControl_U1Em4".manualOperationEmArea[2].displayedLines := '6-13;';
	    "ManualOperationControl_U1Em4".manualOperationEmArea[1].displayedLines := '21-33;';
	END_REGION
	
	REGION Unit 1 Equipment Module 5 configuration
	    "ManualOperationControl_U1Em5".manualOperationEm.equipmentModuleNum := 1060;
	    "ManualOperationControl_U1Em5".manualOperationEmArea[2].displayedLines := '6-13;';
	    "ManualOperationControl_U1Em5".manualOperationEmArea[1].displayedLines := '21-33;';
	END_REGION
	
	REGION Unit 1 Equipment Module 6 configuration
	    "ManualOperationControl_U1Em6".manualOperationEm.equipmentModuleNum := 1070;
	    "ManualOperationControl_U1Em6".manualOperationEmArea[2].displayedLines := '6-18;';
	    "ManualOperationControl_U1Em6".manualOperationEmArea[1].displayedLines := '21-26;';
	END_REGION
	
	REGION Unit 1 Equipment Module 7 configuration
	    "ManualOperationControl_U1Em7".manualOperationEm.equipmentModuleNum := 1080;
	    "ManualOperationControl_U1Em7".manualOperationEmArea[2].displayedLines := '6-14;';
	    "ManualOperationControl_U1Em7".manualOperationEmArea[1].displayedLines := '21-30;';
	END_REGION
	
	REGION CITI EM1 configuration
	    // Statement section REGION
	    "ManualOperationControl_CITIEm1".manualOperationEm.equipmentModuleNum := 5010;
	    "ManualOperationControl_CITIEm1".manualOperationEmArea[1].displayedLines := '1-5;';
	END_REGION
	
END_FUNCTION

FUNCTION "CallManualOperationLines_CITI" : Void   // FC183, LAD
// stored: Access Published, SetENOAutomatically false
   VAR_TEMP
      status : Array[0..30] of Word;   // Status of the Blocks
      errorID : Array[0..30] of Word;   // Error IDs of the Blocks
      call_index : Int;
   END_VAR
   VAR CONSTANT
      MECHANIC_NAME_ENABLE : Bool := FALSE;   // Activation of the Mechanic names
   END_VAR
BEGIN

REGION Network 1: CITI Manual Lines Configuration
   // Equipment Module 3400
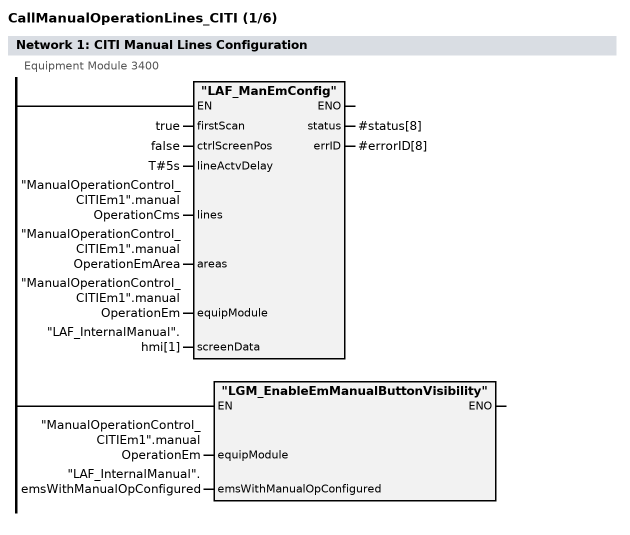
   RUNG wire#powerrail
      "LAF_ManEmConfig"(firstScan := true, ctrlScreenPos := false, lineActvDelay := T#5s, lines := "ManualOperationControl_CITIEm1".manualOperationCms, areas := "ManualOperationControl_CITIEm1".manualOperationEmArea, equipModule := "ManualOperationControl_CITIEm1".manualOperationEm, screenData := "LAF_InternalManual".hmi[1], status => #status[8], errID => #errorID[8])
   END_RUNG
   RUNG wire#powerrail
      "LGM_EnableEmManualButtonVisibility"(equipModule := "ManualOperationControl_CITIEm1".manualOperationEm, emsWithManualOpConfigured := "LAF_InternalManual".emsWithManualOpConfigured)
   END_RUNG
   // the same network as SCL:
   "LAF_ManEmConfig"(firstScan := true,
                     ctrlScreenPos := false,
                     lineActvDelay := T#5s,
                     lines := "ManualOperationControl_CITIEm1".manualOperationCms,
                     areas := "ManualOperationControl_CITIEm1".manualOperationEmArea,
                     equipModule := "ManualOperationControl_CITIEm1".manualOperationEm,
                     screenData := "LAF_InternalManual".hmi[1],
                     status => #status[8],
                     errID => #errorID[8]);
   "LGM_EnableEmManualButtonVisibility"(equipModule := "ManualOperationControl_CITIEm1".manualOperationEm,
                           emsWithManualOpConfigured := "LAF_InternalManual".emsWithManualOpConfigured);
END_REGION

REGION Network 2: CITI1 Equipment Module 1 Line 1
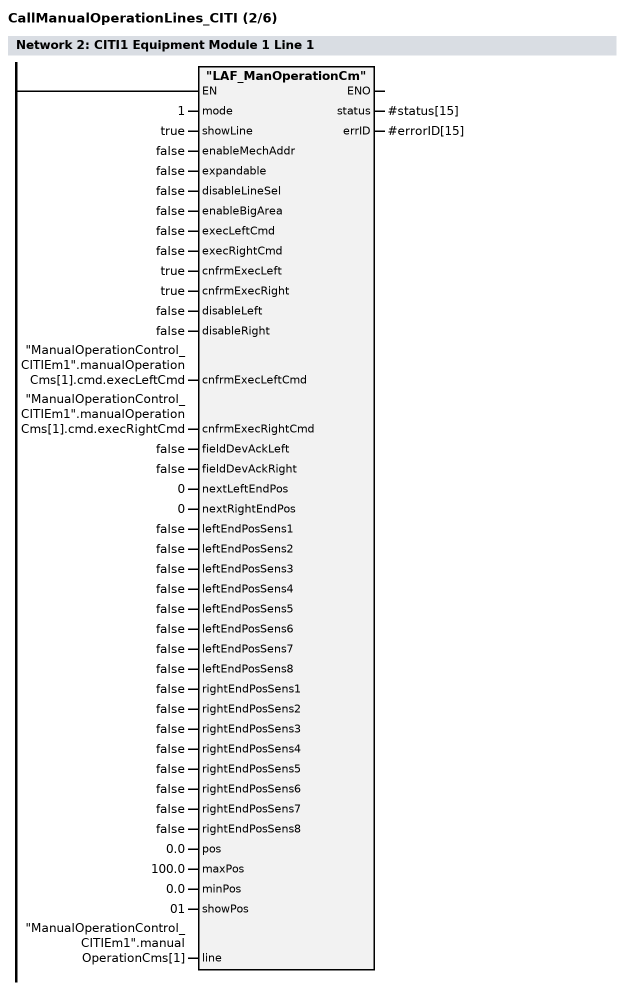
   RUNG wire#powerrail
      "LAF_ManOperationCm"(mode := 1, showLine := true, enableMechAddr := false, expandable := false, disableLineSel := false, enableBigArea := false, execLeftCmd := false, execRightCmd := false, cnfrmExecLeft := true, cnfrmExecRight := true, disableLeft := false, disableRight := false, cnfrmExecLeftCmd := "ManualOperationControl_CITIEm1".manualOperationCms[1].cmd.execLeftCmd, cnfrmExecRightCmd := "ManualOperationControl_CITIEm1".manualOperationCms[1].cmd.execRightCmd, fieldDevAckLeft := false, fieldDevAckRight := false, nextLeftEndPos := 0, nextRightEndPos := 0, leftEndPosSens1 := false, leftEndPosSens2 := false, leftEndPosSens3 := false, leftEndPosSens4 := false, leftEndPosSens5 := false, leftEndPosSens6 := false, leftEndPosSens7 := false, leftEndPosSens8 := false, rightEndPosSens1 := false, rightEndPosSens2 := false, rightEndPosSens3 := false, rightEndPosSens4 := false, rightEndPosSens5 := false, rightEndPosSens6 := false, rightEndPosSens7 := false, rightEndPosSens8 := false, pos := 0.0, maxPos := 100.0, minPos := 0.0, showPos := 01, line := "ManualOperationControl_CITIEm1".manualOperationCms[1], status => #status[15], errID => #errorID[15])
   END_RUNG
   // the same network as SCL:
   "LAF_ManOperationCm"(mode := 1,
                        showLine := true,
                        enableMechAddr := false,
                        expandable := false,
                        disableLineSel := false,
                        enableBigArea := false,
                        execLeftCmd := false,
                        execRightCmd := false,
                        cnfrmExecLeft := true,
                        cnfrmExecRight := true,
                        disableLeft := false,
                        disableRight := false,
                        cnfrmExecLeftCmd := "ManualOperationControl_CITIEm1".manualOperationCms[1].cmd.execLeftCmd,
                        cnfrmExecRightCmd := "ManualOperationControl_CITIEm1".manualOperationCms[1].cmd.execRightCmd,
                        fieldDevAckLeft := false,
                        fieldDevAckRight := false,
                        nextLeftEndPos := 0,
                        nextRightEndPos := 0,
                        leftEndPosSens1 := false,
                        leftEndPosSens2 := false,
                        leftEndPosSens3 := false,
                        leftEndPosSens4 := false,
                        leftEndPosSens5 := false,
                        leftEndPosSens6 := false,
                        leftEndPosSens7 := false,
                        leftEndPosSens8 := false,
                        rightEndPosSens1 := false,
                        rightEndPosSens2 := false,
                        rightEndPosSens3 := false,
                        rightEndPosSens4 := false,
                        rightEndPosSens5 := false,
                        rightEndPosSens6 := false,
                        rightEndPosSens7 := false,
                        rightEndPosSens8 := false,
                        pos := 0.0,
                        maxPos := 100.0,
                        minPos := 0.0,
                        showPos := 01,
                        line := "ManualOperationControl_CITIEm1".manualOperationCms[1],
                        status => #status[15],
                        errID => #errorID[15]);
END_REGION

REGION Network 3: CITI1 Equipment Module 1 Line 2
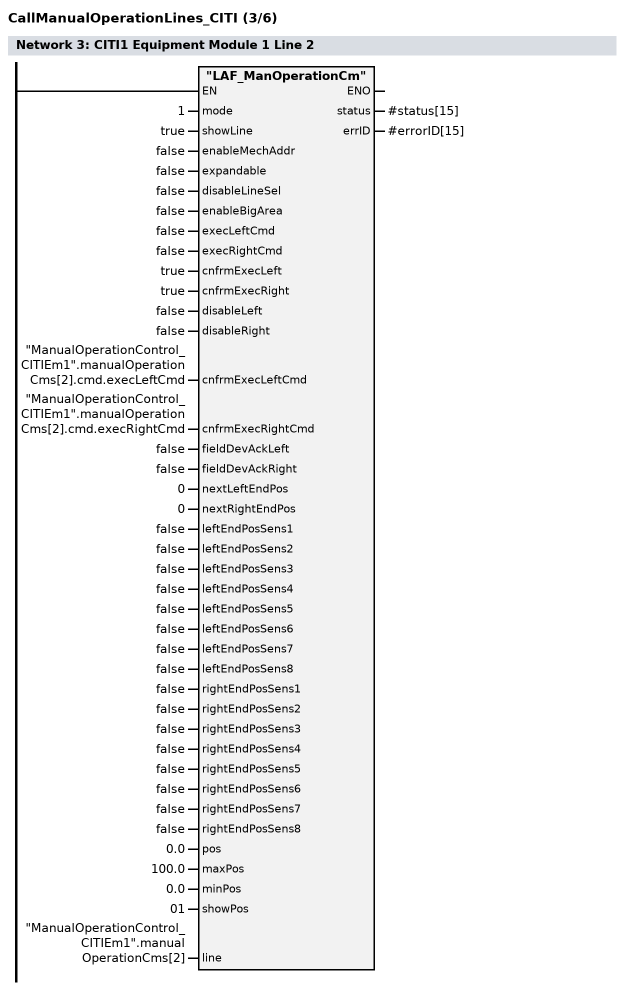
   RUNG wire#powerrail
      "LAF_ManOperationCm"(mode := 1, showLine := true, enableMechAddr := false, expandable := false, disableLineSel := false, enableBigArea := false, execLeftCmd := false, execRightCmd := false, cnfrmExecLeft := true, cnfrmExecRight := true, disableLeft := false, disableRight := false, cnfrmExecLeftCmd := "ManualOperationControl_CITIEm1".manualOperationCms[2].cmd.execLeftCmd, cnfrmExecRightCmd := "ManualOperationControl_CITIEm1".manualOperationCms[2].cmd.execRightCmd, fieldDevAckLeft := false, fieldDevAckRight := false, nextLeftEndPos := 0, nextRightEndPos := 0, leftEndPosSens1 := false, leftEndPosSens2 := false, leftEndPosSens3 := false, leftEndPosSens4 := false, leftEndPosSens5 := false, leftEndPosSens6 := false, leftEndPosSens7 := false, leftEndPosSens8 := false, rightEndPosSens1 := false, rightEndPosSens2 := false, rightEndPosSens3 := false, rightEndPosSens4 := false, rightEndPosSens5 := false, rightEndPosSens6 := false, rightEndPosSens7 := false, rightEndPosSens8 := false, pos := 0.0, maxPos := 100.0, minPos := 0.0, showPos := 01, line := "ManualOperationControl_CITIEm1".manualOperationCms[2], status => #status[15], errID => #errorID[15])
   END_RUNG
   // the same network as SCL:
   "LAF_ManOperationCm"(mode := 1,
                        showLine := true,
                        enableMechAddr := false,
                        expandable := false,
                        disableLineSel := false,
                        enableBigArea := false,
                        execLeftCmd := false,
                        execRightCmd := false,
                        cnfrmExecLeft := true,
                        cnfrmExecRight := true,
                        disableLeft := false,
                        disableRight := false,
                        cnfrmExecLeftCmd := "ManualOperationControl_CITIEm1".manualOperationCms[2].cmd.execLeftCmd,
                        cnfrmExecRightCmd := "ManualOperationControl_CITIEm1".manualOperationCms[2].cmd.execRightCmd,
                        fieldDevAckLeft := false,
                        fieldDevAckRight := false,
                        nextLeftEndPos := 0,
                        nextRightEndPos := 0,
                        leftEndPosSens1 := false,
                        leftEndPosSens2 := false,
                        leftEndPosSens3 := false,
                        leftEndPosSens4 := false,
                        leftEndPosSens5 := false,
                        leftEndPosSens6 := false,
                        leftEndPosSens7 := false,
                        leftEndPosSens8 := false,
                        rightEndPosSens1 := false,
                        rightEndPosSens2 := false,
                        rightEndPosSens3 := false,
                        rightEndPosSens4 := false,
                        rightEndPosSens5 := false,
                        rightEndPosSens6 := false,
                        rightEndPosSens7 := false,
                        rightEndPosSens8 := false,
                        pos := 0.0,
                        maxPos := 100.0,
                        minPos := 0.0,
                        showPos := 01,
                        line := "ManualOperationControl_CITIEm1".manualOperationCms[2],
                        status => #status[15],
                        errID => #errorID[15]);
END_REGION

REGION Network 4: CITI1 Equipment Module 1 Line 3
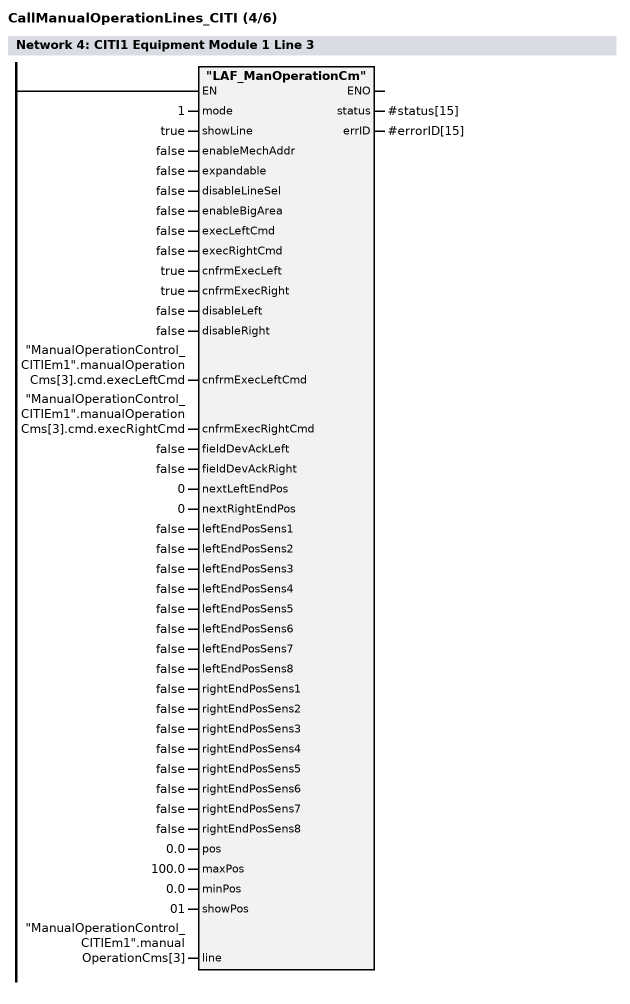
   RUNG wire#powerrail
      "LAF_ManOperationCm"(mode := 1, showLine := true, enableMechAddr := false, expandable := false, disableLineSel := false, enableBigArea := false, execLeftCmd := false, execRightCmd := false, cnfrmExecLeft := true, cnfrmExecRight := true, disableLeft := false, disableRight := false, cnfrmExecLeftCmd := "ManualOperationControl_CITIEm1".manualOperationCms[3].cmd.execLeftCmd, cnfrmExecRightCmd := "ManualOperationControl_CITIEm1".manualOperationCms[3].cmd.execRightCmd, fieldDevAckLeft := false, fieldDevAckRight := false, nextLeftEndPos := 0, nextRightEndPos := 0, leftEndPosSens1 := false, leftEndPosSens2 := false, leftEndPosSens3 := false, leftEndPosSens4 := false, leftEndPosSens5 := false, leftEndPosSens6 := false, leftEndPosSens7 := false, leftEndPosSens8 := false, rightEndPosSens1 := false, rightEndPosSens2 := false, rightEndPosSens3 := false, rightEndPosSens4 := false, rightEndPosSens5 := false, rightEndPosSens6 := false, rightEndPosSens7 := false, rightEndPosSens8 := false, pos := 0.0, maxPos := 100.0, minPos := 0.0, showPos := 01, line := "ManualOperationControl_CITIEm1".manualOperationCms[3], status => #status[15], errID => #errorID[15])
   END_RUNG
   // the same network as SCL:
   "LAF_ManOperationCm"(mode := 1,
                        showLine := true,
                        enableMechAddr := false,
                        expandable := false,
                        disableLineSel := false,
                        enableBigArea := false,
                        execLeftCmd := false,
                        execRightCmd := false,
                        cnfrmExecLeft := true,
                        cnfrmExecRight := true,
                        disableLeft := false,
                        disableRight := false,
                        cnfrmExecLeftCmd := "ManualOperationControl_CITIEm1".manualOperationCms[3].cmd.execLeftCmd,
                        cnfrmExecRightCmd := "ManualOperationControl_CITIEm1".manualOperationCms[3].cmd.execRightCmd,
                        fieldDevAckLeft := false,
                        fieldDevAckRight := false,
                        nextLeftEndPos := 0,
                        nextRightEndPos := 0,
                        leftEndPosSens1 := false,
                        leftEndPosSens2 := false,
                        leftEndPosSens3 := false,
                        leftEndPosSens4 := false,
                        leftEndPosSens5 := false,
                        leftEndPosSens6 := false,
                        leftEndPosSens7 := false,
                        leftEndPosSens8 := false,
                        rightEndPosSens1 := false,
                        rightEndPosSens2 := false,
                        rightEndPosSens3 := false,
                        rightEndPosSens4 := false,
                        rightEndPosSens5 := false,
                        rightEndPosSens6 := false,
                        rightEndPosSens7 := false,
                        rightEndPosSens8 := false,
                        pos := 0.0,
                        maxPos := 100.0,
                        minPos := 0.0,
                        showPos := 01,
                        line := "ManualOperationControl_CITIEm1".manualOperationCms[3],
                        status => #status[15],
                        errID => #errorID[15]);
END_REGION

REGION Network 5: CITI1 Equipment Module 1 Line 4
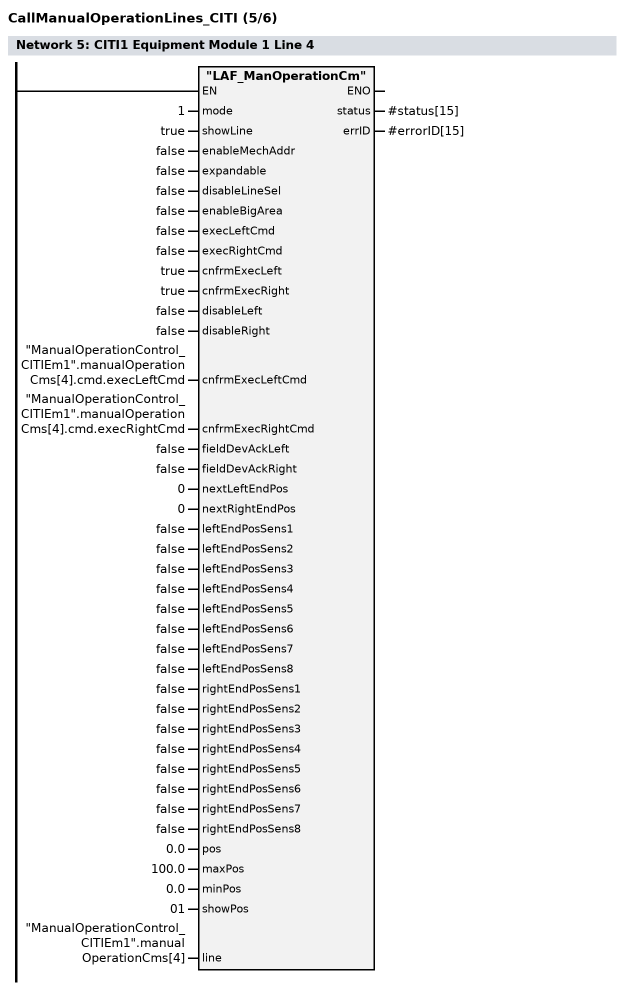
   RUNG wire#powerrail
      "LAF_ManOperationCm"(mode := 1, showLine := true, enableMechAddr := false, expandable := false, disableLineSel := false, enableBigArea := false, execLeftCmd := false, execRightCmd := false, cnfrmExecLeft := true, cnfrmExecRight := true, disableLeft := false, disableRight := false, cnfrmExecLeftCmd := "ManualOperationControl_CITIEm1".manualOperationCms[4].cmd.execLeftCmd, cnfrmExecRightCmd := "ManualOperationControl_CITIEm1".manualOperationCms[4].cmd.execRightCmd, fieldDevAckLeft := false, fieldDevAckRight := false, nextLeftEndPos := 0, nextRightEndPos := 0, leftEndPosSens1 := false, leftEndPosSens2 := false, leftEndPosSens3 := false, leftEndPosSens4 := false, leftEndPosSens5 := false, leftEndPosSens6 := false, leftEndPosSens7 := false, leftEndPosSens8 := false, rightEndPosSens1 := false, rightEndPosSens2 := false, rightEndPosSens3 := false, rightEndPosSens4 := false, rightEndPosSens5 := false, rightEndPosSens6 := false, rightEndPosSens7 := false, rightEndPosSens8 := false, pos := 0.0, maxPos := 100.0, minPos := 0.0, showPos := 01, line := "ManualOperationControl_CITIEm1".manualOperationCms[4], status => #status[15], errID => #errorID[15])
   END_RUNG
   // the same network as SCL:
   "LAF_ManOperationCm"(mode := 1,
                        showLine := true,
                        enableMechAddr := false,
                        expandable := false,
                        disableLineSel := false,
                        enableBigArea := false,
                        execLeftCmd := false,
                        execRightCmd := false,
                        cnfrmExecLeft := true,
                        cnfrmExecRight := true,
                        disableLeft := false,
                        disableRight := false,
                        cnfrmExecLeftCmd := "ManualOperationControl_CITIEm1".manualOperationCms[4].cmd.execLeftCmd,
                        cnfrmExecRightCmd := "ManualOperationControl_CITIEm1".manualOperationCms[4].cmd.execRightCmd,
                        fieldDevAckLeft := false,
                        fieldDevAckRight := false,
                        nextLeftEndPos := 0,
                        nextRightEndPos := 0,
                        leftEndPosSens1 := false,
                        leftEndPosSens2 := false,
                        leftEndPosSens3 := false,
                        leftEndPosSens4 := false,
                        leftEndPosSens5 := false,
                        leftEndPosSens6 := false,
                        leftEndPosSens7 := false,
                        leftEndPosSens8 := false,
                        rightEndPosSens1 := false,
                        rightEndPosSens2 := false,
                        rightEndPosSens3 := false,
                        rightEndPosSens4 := false,
                        rightEndPosSens5 := false,
                        rightEndPosSens6 := false,
                        rightEndPosSens7 := false,
                        rightEndPosSens8 := false,
                        pos := 0.0,
                        maxPos := 100.0,
                        minPos := 0.0,
                        showPos := 01,
                        line := "ManualOperationControl_CITIEm1".manualOperationCms[4],
                        status => #status[15],
                        errID => #errorID[15]);
END_REGION

REGION Network 6: CITI1 Equipment Module 1 Line 5
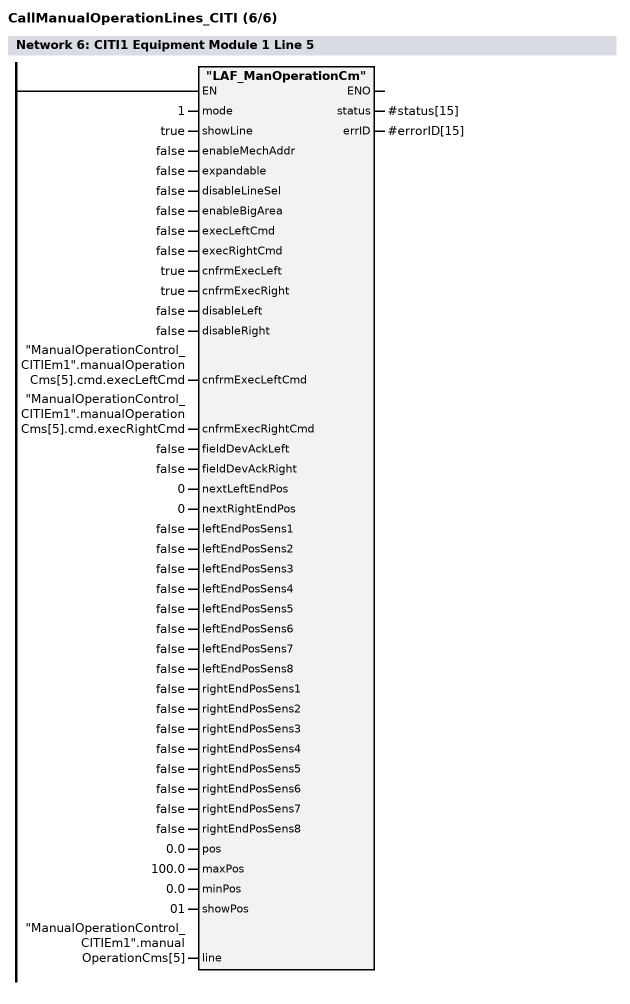
   RUNG wire#powerrail
      "LAF_ManOperationCm"(mode := 1, showLine := true, enableMechAddr := false, expandable := false, disableLineSel := false, enableBigArea := false, execLeftCmd := false, execRightCmd := false, cnfrmExecLeft := true, cnfrmExecRight := true, disableLeft := false, disableRight := false, cnfrmExecLeftCmd := "ManualOperationControl_CITIEm1".manualOperationCms[5].cmd.execLeftCmd, cnfrmExecRightCmd := "ManualOperationControl_CITIEm1".manualOperationCms[5].cmd.execRightCmd, fieldDevAckLeft := false, fieldDevAckRight := false, nextLeftEndPos := 0, nextRightEndPos := 0, leftEndPosSens1 := false, leftEndPosSens2 := false, leftEndPosSens3 := false, leftEndPosSens4 := false, leftEndPosSens5 := false, leftEndPosSens6 := false, leftEndPosSens7 := false, leftEndPosSens8 := false, rightEndPosSens1 := false, rightEndPosSens2 := false, rightEndPosSens3 := false, rightEndPosSens4 := false, rightEndPosSens5 := false, rightEndPosSens6 := false, rightEndPosSens7 := false, rightEndPosSens8 := false, pos := 0.0, maxPos := 100.0, minPos := 0.0, showPos := 01, line := "ManualOperationControl_CITIEm1".manualOperationCms[5], status => #status[15], errID => #errorID[15])
   END_RUNG
   // the same network as SCL:
   "LAF_ManOperationCm"(mode := 1,
                        showLine := true,
                        enableMechAddr := false,
                        expandable := false,
                        disableLineSel := false,
                        enableBigArea := false,
                        execLeftCmd := false,
                        execRightCmd := false,
                        cnfrmExecLeft := true,
                        cnfrmExecRight := true,
                        disableLeft := false,
                        disableRight := false,
                        cnfrmExecLeftCmd := "ManualOperationControl_CITIEm1".manualOperationCms[5].cmd.execLeftCmd,
                        cnfrmExecRightCmd := "ManualOperationControl_CITIEm1".manualOperationCms[5].cmd.execRightCmd,
                        fieldDevAckLeft := false,
                        fieldDevAckRight := false,
                        nextLeftEndPos := 0,
                        nextRightEndPos := 0,
                        leftEndPosSens1 := false,
                        leftEndPosSens2 := false,
                        leftEndPosSens3 := false,
                        leftEndPosSens4 := false,
                        leftEndPosSens5 := false,
                        leftEndPosSens6 := false,
                        leftEndPosSens7 := false,
                        leftEndPosSens8 := false,
                        rightEndPosSens1 := false,
                        rightEndPosSens2 := false,
                        rightEndPosSens3 := false,
                        rightEndPosSens4 := false,
                        rightEndPosSens5 := false,
                        rightEndPosSens6 := false,
                        rightEndPosSens7 := false,
                        rightEndPosSens8 := false,
                        pos := 0.0,
                        maxPos := 100.0,
                        minPos := 0.0,
                        showPos := 01,
                        line := "ManualOperationControl_CITIEm1".manualOperationCms[5],
                        status => #status[15],
                        errID => #errorID[15]);
END_REGION
END_FUNCTION

FUNCTION "LAF_ManualOperationLine_Notes" : Void   // FC23, LAD
TITLE = LAF_ManualOperationLine_Notes
// Here are some points that are important for the use and configuration of manual operation lines:
// 
// * For the appearance of each Line, Json files with the configurations need to be added manually to the target machine. Be it in a PC Runtime or Panel. The Path is set in the HMI as the HMI Tag "manualOperationFilePath" in the "03_manualOperation" table. We have set it to "D:\\JsonFiles\\". The files used for this example are saved in the project UserFiles. The Path for the Panel can look like "/home/industrial/JsonFiles".
// 
// * Under "CallManualOperationLines" are the calls for the main configuration of a Equipment module and the control of each line.
//  * Each Equipment module needs to have a defined number. For the numeration we recommend using the second and third digit for the Equipment module number used in the project and the fourth digit with the number of the unit.
// 
// * The texts for the Areas are defined as text lists in the HMI. For the corresponding group, the naming is currently set as "EquipmentAreas_XXXX" with the XXXX as the Equipment Module number. It is set in the "manualOperationEm.equipmentModuleNum".
//  
// * There can be defined 16 color text lists. Each text list defines: "1 - normal, 2 - pressed, 3 - confirmed, 4 - deactivated, 5 - deactivated+pressed".
//  * The color value is in hex with the 2 first values on the left defining the transparency and the rest as normal color values.
//  * The text list name is currently "LAF_manualColorX" with the X as the text list number.
// 
// * If another HMI device is added, please don't forget the Scheduled tasks for updating the lines  
// 
// * The amount of areas is defined by the size of the array in the configuration of areas. The array should start.
// stored: SetENOAutomatically false
BEGIN
END_FUNCTION

FUNCTION "CallShiftModel" : Void   // FC2, LAD
TITLE = CallShiftModel
// Called LSicar_Shiftmodel
// stored: IsIECCheckEnabled true, SetENOAutomatically true
   VAR_TEMP   // added for the SCL form of the ladder/FBD networks
      _w1 : Bool;
      _w2 : Bool;
      _w3 : Bool;
   END_VAR
BEGIN

REGION Network 1: BLOCK INFO HEADER
   // SIEMENS AG / (c)Copyright 2023
   // ------------------------------------------------------------------------------
   // Title:            CallShiftModel (FC2)
   // Comment/Function: Called LSicar_Shiftmodel 
   // Library/Family:   Automation Framework
   // Author:           Siemens Digital Industry
   // Tested with:      ---
   // Engineering:      TIA Portal V19
   // Restrictions:     -
   // Requirements:     ---
   // ------------------------------------------------------------------------------
   // Change log table:
   // Version  | Date       | Expert in charge       | Changes applied
   // ---------|------------|------------------------|------------------------------
   // 01.00.00 | 11.12.2023 | Siemens Industry Online Support
   //                         First released version
END_REGION

REGION Network 2: Call: shiftmodel
   // FB for handling the shift model and times
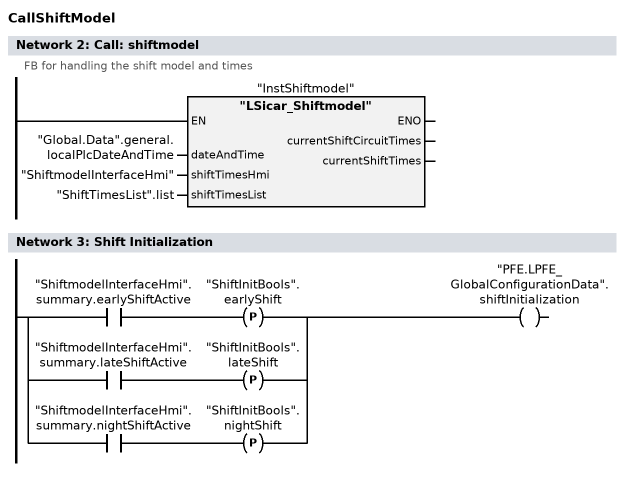
   RUNG wire#powerrail
      "InstShiftmodel"(dateAndTime := "Global.Data".general.localPlcDateAndTime, shiftTimesHmi := "ShiftmodelInterfaceHmi", shiftTimesList := "ShiftTimesList".list, currentShiftCircuitTimes =>, currentShiftTimes =>)
   END_RUNG
   // the same network as SCL:
   "InstShiftmodel"(dateAndTime := "Global.Data".general.localPlcDateAndTime,   // "LSicar_Shiftmodel"
                    shiftTimesHmi := "ShiftmodelInterfaceHmi",
                    shiftTimesList := "ShiftTimesList".list);
END_REGION

REGION Network 3: Shift Initialization
   RUNG wire#powerrail
      Contact( "ShiftmodelInterfaceHmi".summary.earlyShiftActive )
      P_Trig( "ShiftInitBools".earlyShift )
      wire#w1
      Coil( "PFE.LPFE_GlobalConfigurationData".shiftInitialization )
   END_RUNG
   RUNG wire#powerrail
      Contact( "ShiftmodelInterfaceHmi".summary.lateShiftActive )
      P_Trig( "ShiftInitBools".lateShift )
   END_RUNG wire#w1
   RUNG wire#powerrail
      Contact( "ShiftmodelInterfaceHmi".summary.nightShiftActive )
      P_Trig( "ShiftInitBools".nightShift )
   END_RUNG wire#w1
   // the same network as SCL:
   #_w1 := "ShiftmodelInterfaceHmi".summary.earlyShiftActive AND NOT "ShiftInitBools".earlyShift;   // rising edge
   "ShiftInitBools".earlyShift := "ShiftmodelInterfaceHmi".summary.earlyShiftActive;
   #_w2 := "ShiftmodelInterfaceHmi".summary.lateShiftActive AND NOT "ShiftInitBools".lateShift;   // rising edge
   "ShiftInitBools".lateShift := "ShiftmodelInterfaceHmi".summary.lateShiftActive;
   #_w3 := "ShiftmodelInterfaceHmi".summary.nightShiftActive AND NOT "ShiftInitBools".nightShift;   // rising edge
   "ShiftInitBools".nightShift := "ShiftmodelInterfaceHmi".summary.nightShiftActive;
   "PFE.LPFE_GlobalConfigurationData".shiftInitialization := #_w1 OR #_w2 OR #_w3;
END_REGION
END_FUNCTION

FUNCTION "ReadMe01" : Void
{ S7_Optimized_Access := 'TRUE' ; Published := 'FALSE' }
VERSION : 0.1

BEGIN
	// The folder structure of the software unit CentralFunctions correlates with the main navigation in the HMI.
	// For easier orientation, all folders are listed, but some are empty because there is no PLC logic needed, there is only content on the HMI side.
	// Any PLC logic that should relate to the screens on the HMI for that chapter can be added in this folder.
END_FUNCTION

FUNCTION "ReadMe02" : Void
{ S7_Optimized_Access := 'TRUE' ; Published := 'FALSE' }
VERSION : 0.1

BEGIN
	// The folder structure of the software unit CentralFunctions correlates with the main navigation in the HMI.
	// For easier orientation, all folders are listed, but some are empty because there is no PLC logic needed, there is only content on the HMI side.
	// Any PLC logic that should relate to the screens on the HMI for that chapter can be added in this folder.
END_FUNCTION

FUNCTION "CallManualOperationLines_ServoCommands" : Void
{ S7_Optimized_Access := 'TRUE' ; Published := 'FALSE' }
VERSION : 0.1
   VAR_INPUT 
      ManualOperationControl : "LBC_typeAxisControlManualCommands";
   END_VAR

   VAR_OUTPUT 
      HmiInterface : "LBC_typeAxisControlManualCommands";
   END_VAR


BEGIN
	REGION Commands Mapping
	    //#HmiInterface.enableAxis := #ManualOperationControl.enableAxis;
	    //#HmiInterface.resetAxis := #ManualOperationControl.resetAxis;
	    
	    #HmiInterface.jogForward := #ManualOperationControl.jogForward;
	    #HmiInterface.jogBackward := #ManualOperationControl.jogBackward;
	    
	    //#HmiInterface.moveVelocity := #ManualOperationControl.moveVelocity;
	    //#HmiInterface.stop := #ManualOperationControl.stop;
	    //#HmiInterface.posRelative := #ManualOperationControl.posRelative;
	    //#HmiInterface.posAbsolute := #ManualOperationControl.posAbsolute;
	END_REGION
	
END_FUNCTION

FUNCTION "CallManualOperationLines_ServoPos64Commands" : Void
{ S7_Optimized_Access := 'TRUE' ; Published := 'FALSE' }
VERSION : 0.1
   VAR_INPUT 
      ManualOperationControl : "LBC_typeAxis64PosManualCommands";
   END_VAR

   VAR_OUTPUT 
      HmiInterface : "LBC_typeAxis64PosManualCommands";
   END_VAR


BEGIN
	REGION Commands Mapping
	    //#HmiInterface.enableAxis := #ManualOperationControl.enableAxis;
	    //#HmiInterface.resetAxis := #ManualOperationControl.resetAxis;
	    
	    #HmiInterface.jogForward := #ManualOperationControl.jogForward;
	    #HmiInterface.jogBackward := #ManualOperationControl.jogBackward;
	    
	    //#HmiInterface.moveVelocity := #ManualOperationControl.moveVelocity;
	    //#HmiInterface.stop := #ManualOperationControl.stop;
	    //#HmiInterface.posRelative := #ManualOperationControl.posRelative;
	    //#HmiInterface.posAbsolute := #ManualOperationControl.posAbsolute;
	END_REGION
	
END_FUNCTION

FUNCTION "ReadMe04" : Void
{ S7_Optimized_Access := 'TRUE' ; Published := 'FALSE' }
VERSION : 0.1

BEGIN
	// The folder structure of the software unit CentralFunctions correlates with the main navigation in the HMI.
	// For easier orientation, all folders are listed, but some are empty because there is no PLC logic needed, there is only content on the HMI side.
	// Any PLC logic that should relate to the screens on the HMI for that chapter can be added in this folder.
END_FUNCTION

FUNCTION "ReadMe06" : Void
{ S7_Optimized_Access := 'TRUE' ; Published := 'FALSE' }
VERSION : 0.1

BEGIN
	// The folder structure of the software unit CentralFunctions correlates with the main navigation in the HMI.
	// For easier orientation, all folders are listed, but some are empty because there is no PLC logic needed, there is only content on the HMI side.
	// Any PLC logic that should relate to the screens on the HMI for that chapter can be added in this folder.
END_FUNCTION

FUNCTION "ReadMe10" : Void
{ S7_Optimized_Access := 'TRUE' ; Published := 'FALSE' }
VERSION : 0.1

BEGIN
	// The folder structure of the software unit CentralFunctions correlates with the main navigation in the HMI.
	// For easier orientation, all folders are listed, but some are empty because there is no PLC logic needed, there is only content on the HMI side.
	// Any PLC logic that should relate to the screens on the HMI for that chapter can be added in this folder.
END_FUNCTION

FUNCTION "ReadMe11" : Void
{ S7_Optimized_Access := 'TRUE' ; Published := 'FALSE' }
VERSION : 0.1

BEGIN
	// The folder structure of the software unit CentralFunctions correlates with the main navigation in the HMI.
	// For easier orientation, all folders are listed, but some are empty because there is no PLC logic needed, there is only content on the HMI side.
	// Any PLC logic that should relate to the screens on the HMI for that chapter can be added in this folder.
END_FUNCTION

DATA_BLOCK "LER_Recipe_DB"   // DB116
// stored: InstanceOfName LER_Recipe, InstanceOfType FB
"LER_Recipe"
   // VAR_INPUT
   //    enable : Bool;
   //    applyBT : Bool;
   // END_VAR
   // VAR_IN_OUT
   //    parameterRecipeInterface : "HMI_IF_Parameter_LIstRecipe_Interface";
   //    parameterListSV : "HMI_IF_Parameter_ListRecipe_UDT";
   //    parameterListPV : "HMI_IF_Parameter_ListRecipe_UDT";
   // END_VAR
BEGIN
END_DATA_BLOCK

DATA_BLOCK "instTeachingPosJRPusherAxisZ"   // DB134
// stored: InstanceOfName LER_TeachingPos_Interface, InstanceOfType FB
"LER_TeachingPos_Interface"
   // VAR_INPUT
   //    enable : Bool;
   //    selectTeachingPos : SInt;
   //    indexTeachingPos : SInt;
   // END_VAR
   // VAR_IN_OUT
   //    configurationSetPositions : Array[0..15] of "LBC_typeAxis64PosSetPosition";
   //    moduleInterface : "LBC_typeAxis64PosInterface";
   //    hmiInterface : Array[0..48] of "LER_TypeTeachingPosInterface";
   // END_VAR
   // VAR
   //    statPulse : Array[0..9] of Bool;
   //    statTonTimer : Array[0..15] of TON_TIME;
   //    statLastTeachingPosIndex : SInt;
   // END_VAR
BEGIN
END_DATA_BLOCK

DATA_BLOCK "InstCallAlarmCounter"   // DB25
// stored: InstanceOfName CallAlarmCounter, InstanceOfType FB
"CallAlarmCounter"
BEGIN
END_DATA_BLOCK

DATA_BLOCK "InstCallProcessCount"   // DB24
// stored: InstanceOfName CallProcessCount, InstanceOfType FB
"CallProcessCount"
BEGIN
END_DATA_BLOCK

